	VAR robtarget Openhole_694 := [[468.83, -10.99, 179.55], [0.039839, 0.705984, 0.70118, -0.091361], [0,0,0,0], [9E9, 9E9, 9E9, 9E9, 9E9, 9E9]];
	VAR robtarget Openhole_695 := [[469.79, -10.75, 179.43], [0.042242, 0.705844, 0.700663, -0.095246], [0,0,0,0], [9E9, 9E9, 9E9, 9E9, 9E9, 9E9]];
	VAR robtarget Openhole_696 := [[473.7, -10.06, 178.96], [0.052829, 0.705131, 0.698512, -0.109911], [0,0,0,0], [9E9, 9E9, 9E9, 9E9, 9E9, 9E9]];
	VAR robtarget Openhole_697 := [[478.16, -9.69, 178.47], [0.066049, 0.704015, 0.695989, -0.124897], [0,0,0,0], [9E9, 9E9, 9E9, 9E9, 9E9, 9E9]];
	VAR robtarget Openhole_698 := [[482.14, -9.61, 178.09], [0.078462, 0.70274, 0.693688, -0.137102], [0,0,0,0], [9E9, 9E9, 9E9, 9E9, 9E9, 9E9]];
	VAR robtarget Openhole_699 := [[482.63, -9.62, 178.05], [0.080033, 0.702563, 0.693396, -0.13857], [0,0,0,0], [9E9, 9E9, 9E9, 9E9, 9E9, 9E9]];
	VAR robtarget Openhole_700 := [[494.09, -10.02, 177.18], [0.116014, 0.697525, 0.686428, -0.169755], [0,0,0,0], [9E9, 9E9, 9E9, 9E9, 9E9, 9E9]];
	VAR robtarget Openhole_701 := [[499.58, -10.13, 176.76], [0.132008, 0.694675, 0.682777, -0.183891], [0,0,0,0], [9E9, 9E9, 9E9, 9E9, 9E9, 9E9]];
	VAR robtarget Openhole_702 := [[500.07, -10.12, 176.71], [0.133393, 0.694411, 0.682429, -0.185176], [0,0,0,0], [9E9, 9E9, 9E9, 9E9, 9E9, 9E9]];
	VAR robtarget Openhole_703 := [[503.55, -10.02, 176.36], [0.142648, 0.692569, 0.6799, -0.194257], [0,0,0,0], [9E9, 9E9, 9E9, 9E9, 9E9, 9E9]];
	VAR robtarget Openhole_704 := [[504.33, -10, 176.29], [0.144708, 0.692141, 0.679339, -0.196212], [0,0,0,0], [9E9, 9E9, 9E9, 9E9, 9E9, 9E9]];
	VAR robtarget Openhole_705 := [[509.33, -10, 175.85], [0.183051, 0.683002, 0.683002, -0.183051], [0,0,0,0], [9E9, 9E9, 9E9, 9E9, 9E9, 9E9]];
	VAR robtarget Openhole_706 := [[536.33, -10, 175.77], [0.183051, 0.683002, 0.683002, -0.183051], [0,0,0,0], [9E9, 9E9, 9E9, 9E9, 9E9, 9E9]];
	VAR robtarget Openhole_707 := [[536.33, -10.89, 176.28], [0.183051, 0.683002, 0.683002, -0.183051], [0,0,0,0], [9E9, 9E9, 9E9, 9E9, 9E9, 9E9]];
	VAR robtarget Openhole_708 := [[524.33, -10.89, 176.31], [0.183051, 0.683002, 0.683002, -0.183051], [0,0,0,0], [9E9, 9E9, 9E9, 9E9, 9E9, 9E9]];
	VAR robtarget Openhole_709 := [[509.33, -10.89, 176.36], [0.183051, 0.683002, 0.683002, -0.183051], [0,0,0,0], [9E9, 9E9, 9E9, 9E9, 9E9, 9E9]];
	VAR robtarget Openhole_710 := [[504.39, -10.89, 176.75], [0.147452, 0.691562, 0.680025, -0.19382], [0,0,0,0], [9E9, 9E9, 9E9, 9E9, 9E9, 9E9]];
	VAR robtarget Openhole_711 := [[498.87, -11.14, 177.3], [0.13304, 0.694478, 0.684057, -0.179068], [0,0,0,0], [9E9, 9E9, 9E9, 9E9, 9E9, 9E9]];
	VAR robtarget Openhole_712 := [[497.37, -11.14, 177.42], [0.12885, 0.695268, 0.685077, -0.175125], [0,0,0,0], [9E9, 9E9, 9E9, 9E9, 9E9, 9E9]];
	VAR robtarget Openhole_713 := [[496.87, -11.14, 177.45], [0.127427, 0.69553, 0.685411, -0.173814], [0,0,0,0], [9E9, 9E9, 9E9, 9E9, 9E9, 9E9]];
	VAR robtarget Openhole_714 := [[482.41, -10.79, 178.44], [0.083092, 0.702208, 0.69426, -0.134176], [0,0,0,0], [9E9, 9E9, 9E9, 9E9, 9E9, 9E9]];
	VAR robtarget Openhole_715 := [[481.91, -10.8, 178.48], [0.081533, 0.70239, 0.694546, -0.132689], [0,0,0,0], [9E9, 9E9, 9E9, 9E9, 9E9, 9E9]];
	VAR robtarget Openhole_716 := [[476.44, -10.97, 178.96], [0.064669, 0.704143, 0.69761, -0.115499], [0,0,0,0], [9E9, 9E9, 9E9, 9E9, 9E9, 9E9]];
	VAR robtarget Openhole_717 := [[472.49, -11.44, 179.37], [0.053367, 0.70509, 0.699769, -0.101607], [0,0,0,0], [9E9, 9E9, 9E9, 9E9, 9E9, 9E9]];
	VAR robtarget Openhole_718 := [[471.02, -11.7, 179.53], [0.049411, 0.705378, 0.700549, -0.096078], [0,0,0,0], [9E9, 9E9, 9E9, 9E9, 9E9, 9E9]];
	VAR robtarget Openhole_719 := [[470.53, -11.8, 179.59], [0.048148, 0.705466, 0.700806, -0.094186], [0,0,0,0], [9E9, 9E9, 9E9, 9E9, 9E9, 9E9]];
	VAR robtarget Openhole_720 := [[469.57, -12.03, 179.7], [0.045713, 0.705628, 0.701314, -0.090326], [0,0,0,0], [9E9, 9E9, 9E9, 9E9, 9E9, 9E9]];
	VAR robtarget Openhole_721 := [[468.61, -12.29, 179.81], [0.043403, 0.705773, 0.701812, -0.086369], [0,0,0,0], [9E9, 9E9, 9E9, 9E9, 9E9, 9E9]];
	VAR robtarget Openhole_722 := [[467.66, -12.58, 179.92], [0.041218, 0.705904, 0.702299, -0.08232], [0,0,0,0], [9E9, 9E9, 9E9, 9E9, 9E9, 9E9]];
	VAR robtarget Openhole_723 := [[466.25, -13.07, 180.09], [0.038201, 0.706074, 0.703002, -0.076079], [0,0,0,0], [9E9, 9E9, 9E9, 9E9, 9E9, 9E9]];
	VAR robtarget Openhole_724 := [[465.79, -13.26, 180.15], [0.037278, 0.706123, 0.703229, -0.073951], [0,0,0,0], [9E9, 9E9, 9E9, 9E9, 9E9, 9E9]];
	VAR robtarget Openhole_725 := [[465.33, -13.45, 180.2], [0.036401, 0.706169, 0.703452, -0.071798], [0,0,0,0], [9E9, 9E9, 9E9, 9E9, 9E9, 9E9]];
	VAR robtarget Openhole_726 := [[464.88, -13.66, 180.26], [0.03558, 0.706211, 0.703671, -0.06962], [0,0,0,0], [9E9, 9E9, 9E9, 9E9, 9E9, 9E9]];
	VAR robtarget Openhole_727 := [[463.11, -14.56, 180.47], [0.032691, 0.706351, 0.704495, -0.060722], [0,0,0,0], [9E9, 9E9, 9E9, 9E9, 9E9, 9E9]];
	VAR robtarget Openhole_728 := [[461.82, -15.31, 180.62], [0.030887, 0.706432, 0.70505, -0.053896], [0,0,0,0], [9E9, 9E9, 9E9, 9E9, 9E9, 9E9]];
	VAR robtarget Openhole_729 := [[460.15, -16.4, 180.79], [0.028933, 0.706515, 0.705697, -0.044632], [0,0,0,0], [9E9, 9E9, 9E9, 9E9, 9E9, 9E9]];
	VAR robtarget Openhole_730 := [[459.72, -16.65, 180.82], [0.028341, 0.706539, 0.705839, -0.04233], [0,0,0,0], [9E9, 9E9, 9E9, 9E9, 9E9, 9E9]];
	VAR robtarget Openhole_731 := [[459.27, -16.88, 180.86], [0.027587, 0.706568, 0.70597, -0.040074], [0,0,0,0], [9E9, 9E9, 9E9, 9E9, 9E9, 9E9]];
	VAR robtarget Openhole_732 := [[458.82, -17.08, 180.88], [0.026741, 0.706601, 0.706093, -0.037847], [0,0,0,0], [9E9, 9E9, 9E9, 9E9, 9E9, 9E9]];
	VAR robtarget Openhole_733 := [[458.35, -17.26, 180.91], [0.025788, 0.706636, 0.706207, -0.03566], [0,0,0,0], [9E9, 9E9, 9E9, 9E9, 9E9, 9E9]];
	VAR robtarget Openhole_734 := [[457.88, -17.43, 180.93], [0.024778, 0.706673, 0.706313, -0.033497], [0,0,0,0], [9E9, 9E9, 9E9, 9E9, 9E9, 9E9]];
	VAR robtarget Openhole_735 := [[457.27, -17.6, 180.95], [0.023274, 0.706724, 0.706433, -0.030857], [0,0,0,0], [9E9, 9E9, 9E9, 9E9, 9E9, 9E9]];
	VAR robtarget Openhole_736 := [[454.82, -17.6, 180.99], [0.014998, 0.706948, 0.706747, -0.022558], [0,0,0,0], [9E9, 9E9, 9E9, 9E9, 9E9, 9E9]];
	VAR robtarget Openhole_737 := [[454.9, -18.58, 181.04], [0.018567, 0.706863, 0.706838, -0.019489], [0,0,0,0], [9E9, 9E9, 9E9, 9E9, 9E9, 9E9]];
	VAR robtarget Openhole_738 := [[457.34, -18.58, 181.03], [0.026836, 0.706597, 0.70656, -0.027794], [0,0,0,0], [9E9, 9E9, 9E9, 9E9, 9E9, 9E9]];
	VAR robtarget Openhole_739 := [[457.46, -18.57, 181.03], [0.027232, 0.706582, 0.706544, -0.0282], [0,0,0,0], [9E9, 9E9, 9E9, 9E9, 9E9, 9E9]];
	VAR robtarget Openhole_740 := [[457.96, -18.57, 181.02], [0.028901, 0.706516, 0.706474, -0.029909], [0,0,0,0], [9E9, 9E9, 9E9, 9E9, 9E9, 9E9]];
	VAR robtarget Openhole_741 := [[458.45, -18.46, 181.01], [0.030176, 0.706463, 0.706386, -0.031929], [0,0,0,0], [9E9, 9E9, 9E9, 9E9, 9E9, 9E9]];
	VAR robtarget Openhole_742 := [[459.42, -18.22, 180.98], [0.032613, 0.706354, 0.706188, -0.036029], [0,0,0,0], [9E9, 9E9, 9E9, 9E9, 9E9, 9E9]];
	VAR robtarget Openhole_743 := [[460.37, -17.92, 180.94], [0.03481, 0.706249, 0.70596, -0.040251], [0,0,0,0], [9E9, 9E9, 9E9, 9E9, 9E9, 9E9]];
	VAR robtarget Openhole_744 := [[460.84, -17.74, 180.92], [0.035759, 0.706202, 0.705833, -0.042429], [0,0,0,0], [9E9, 9E9, 9E9, 9E9, 9E9, 9E9]];
	VAR robtarget Openhole_745 := [[461.3, -17.54, 180.89], [0.036653, 0.706156, 0.705697, -0.044628], [0,0,0,0], [9E9, 9E9, 9E9, 9E9, 9E9, 9E9]];
	VAR robtarget Openhole_746 := [[462.19, -17.09, 180.82], [0.038087, 0.70608, 0.705397, -0.049141], [0,0,0,0], [9E9, 9E9, 9E9, 9E9, 9E9, 9E9]];
	VAR robtarget Openhole_747 := [[463.94, -16.14, 180.66], [0.040777, 0.70593, 0.70471, -0.058174], [0,0,0,0], [9E9, 9E9, 9E9, 9E9, 9E9, 9E9]];
	VAR robtarget Openhole_748 := [[464.83, -15.7, 180.57], [0.042243, 0.705844, 0.704328, -0.062628], [0,0,0,0], [9E9, 9E9, 9E9, 9E9, 9E9, 9E9]];
	VAR robtarget Openhole_749 := [[465.73, -15.28, 180.47], [0.043835, 0.705747, 0.703924, -0.067018], [0,0,0,0], [9E9, 9E9, 9E9, 9E9, 9E9, 9E9]];
	VAR robtarget Openhole_750 := [[466.19, -15.08, 180.42], [0.044689, 0.705693, 0.703714, -0.069185], [0,0,0,0], [9E9, 9E9, 9E9, 9E9, 9E9, 9E9]];
	VAR robtarget Openhole_751 := [[466.65, -14.89, 180.37], [0.045584, 0.705636, 0.7035, -0.07133], [0,0,0,0], [9E9, 9E9, 9E9, 9E9, 9E9, 9E9]];
	VAR robtarget Openhole_752 := [[467.12, -14.71, 180.32], [0.046532, 0.705574, 0.703282, -0.073447], [0,0,0,0], [9E9, 9E9, 9E9, 9E9, 9E9, 9E9]];
	VAR robtarget Openhole_753 := [[467.58, -14.54, 180.27], [0.047528, 0.705508, 0.703061, -0.075537], [0,0,0,0], [9E9, 9E9, 9E9, 9E9, 9E9, 9E9]];
	VAR robtarget Openhole_754 := [[468.53, -14.24, 180.18], [0.049641, 0.705362, 0.702607, -0.079642], [0,0,0,0], [9E9, 9E9, 9E9, 9E9, 9E9, 9E9]];
	VAR robtarget Openhole_755 := [[469.49, -13.97, 180.08], [0.0519, 0.7052, 0.702142, -0.083648], [0,0,0,0], [9E9, 9E9, 9E9, 9E9, 9E9, 9E9]];
	VAR robtarget Openhole_756 := [[470.46, -13.73, 179.98], [0.054271, 0.705021, 0.701664, -0.087567], [0,0,0,0], [9E9, 9E9, 9E9, 9E9, 9E9, 9E9]];
	VAR robtarget Openhole_757 := [[470.94, -13.62, 179.94], [0.055498, 0.704925, 0.701421, -0.089491], [0,0,0,0], [9E9, 9E9, 9E9, 9E9, 9E9, 9E9]];
	VAR robtarget Openhole_758 := [[471.92, -13.42, 179.84], [0.058039, 0.704721, 0.700929, -0.093267], [0,0,0,0], [9E9, 9E9, 9E9, 9E9, 9E9, 9E9]];
	VAR robtarget Openhole_759 := [[475.87, -12.91, 179.5], [0.069183, 0.703714, 0.698901, -0.107409], [0,0,0,0], [9E9, 9E9, 9E9, 9E9, 9E9, 9E9]];
	VAR robtarget Openhole_760 := [[480.85, -12.71, 179.15], [0.084353, 0.702057, 0.69626, -0.12338], [0,0,0,0], [9E9, 9E9, 9E9, 9E9, 9E9, 9E9]];
	VAR robtarget Openhole_761 := [[482.35, -12.7, 179.05], [0.088996, 0.701484, 0.69544, -0.127919], [0,0,0,0], [9E9, 9E9, 9E9, 9E9, 9E9, 9E9]];
	VAR robtarget Openhole_762 := [[482.85, -12.7, 179.02], [0.090547, 0.701285, 0.695164, -0.12941], [0,0,0,0], [9E9, 9E9, 9E9, 9E9, 9E9, 9E9]];
	VAR robtarget Openhole_763 := [[495.33, -12.89, 178.35], [0.12834, 0.695362, 0.687731, -0.164398], [0,0,0,0], [9E9, 9E9, 9E9, 9E9, 9E9, 9E9]];
	VAR robtarget Openhole_764 := [[495.83, -12.89, 178.32], [0.129759, 0.695099, 0.687406, -0.165751], [0,0,0,0], [9E9, 9E9, 9E9, 9E9, 9E9, 9E9]];
	VAR robtarget Openhole_765 := [[501.81, -12.75, 177.89], [0.145951, 0.69188, 0.683309, -0.181905], [0,0,0,0], [9E9, 9E9, 9E9, 9E9, 9E9, 9E9]];
	VAR robtarget Openhole_766 := [[504.33, -12.58, 177.65], [0.152252, 0.690521, 0.681443, -0.188774], [0,0,0,0], [9E9, 9E9, 9E9, 9E9, 9E9, 9E9]];
	VAR robtarget Openhole_767 := [[509.33, -12.58, 177.34], [0.183051, 0.683002, 0.683002, -0.183051], [0,0,0,0], [9E9, 9E9, 9E9, 9E9, 9E9, 9E9]];
	VAR robtarget Openhole_768 := [[536.33, -12.58, 177.26], [0.183051, 0.683002, 0.683002, -0.183051], [0,0,0,0], [9E9, 9E9, 9E9, 9E9, 9E9, 9E9]];
	VAR robtarget Openhole_769 := [[536.34, -16.49, 179.51], [0.183051, 0.683002, 0.683002, -0.183051], [0,0,0,0], [9E9, 9E9, 9E9, 9E9, 9E9, 9E9]];
	VAR robtarget Openhole_770 := [[509.34, -16.49, 179.6], [0.183051, 0.683002, 0.683002, -0.183051], [0,0,0,0], [9E9, 9E9, 9E9, 9E9, 9E9, 9E9]];
	VAR robtarget Openhole_771 := [[504.34, -16.49, 179.72], [0.163682, 0.687901, 0.684485, -0.177427], [0,0,0,0], [9E9, 9E9, 9E9, 9E9, 9E9, 9E9]];
	VAR robtarget Openhole_772 := [[497.74, -16.81, 180.03], [0.146949, 0.691669, 0.688969, -0.159127], [0,0,0,0], [9E9, 9E9, 9E9, 9E9, 9E9, 9E9]];
	VAR robtarget Openhole_773 := [[491.74, -16.89, 180.19], [0.130322, 0.694994, 0.692656, -0.142222], [0,0,0,0], [9E9, 9E9, 9E9, 9E9, 9E9, 9E9]];
	VAR robtarget Openhole_774 := [[491.24, -16.89, 180.2], [0.12888, 0.695263, 0.692947, -0.140799], [0,0,0,0], [9E9, 9E9, 9E9, 9E9, 9E9, 9E9]];
	VAR robtarget Openhole_775 := [[478.25, -16.73, 180.42], [0.08917, 0.701462, 0.699653, -0.102403], [0,0,0,0], [9E9, 9E9, 9E9, 9E9, 9E9, 9E9]];
	VAR robtarget Openhole_776 := [[477.75, -16.74, 180.44], [0.087603, 0.701659, 0.69988, -0.100837], [0,0,0,0], [9E9, 9E9, 9E9, 9E9, 9E9, 9E9]];
	VAR robtarget Openhole_777 := [[472.25, -16.88, 180.59], [0.070529, 0.703581, 0.702227, -0.082932], [0,0,0,0], [9E9, 9E9, 9E9, 9E9, 9E9, 9E9]];
	VAR robtarget Openhole_778 := [[471.26, -16.95, 180.62], [0.067552, 0.703873, 0.702627, -0.079465], [0,0,0,0], [9E9, 9E9, 9E9, 9E9, 9E9, 9E9]];
	VAR robtarget Openhole_779 := [[470.26, -17.06, 180.67], [0.064687, 0.704142, 0.703023, -0.075881], [0,0,0,0], [9E9, 9E9, 9E9, 9E9, 9E9, 9E9]];
	VAR robtarget Openhole_780 := [[468.29, -17.35, 180.76], [0.05919, 0.704625, 0.703785, -0.06846], [0,0,0,0], [9E9, 9E9, 9E9, 9E9, 9E9, 9E9]];
	VAR robtarget Openhole_781 := [[467.79, -17.44, 180.78], [0.057875, 0.704734, 0.703968, -0.06655], [0,0,0,0], [9E9, 9E9, 9E9, 9E9, 9E9, 9E9]];
	VAR robtarget Openhole_782 := [[467.31, -17.54, 180.8], [0.056598, 0.704838, 0.704149, -0.064606], [0,0,0,0], [9E9, 9E9, 9E9, 9E9, 9E9, 9E9]];
	VAR robtarget Openhole_783 := [[465.37, -18.02, 180.91], [0.05178, 0.705208, 0.704838, -0.056602], [0,0,0,0], [9E9, 9E9, 9E9, 9E9, 9E9, 9E9]];
	VAR robtarget Openhole_784 := [[464.4, -18.28, 180.95], [0.049485, 0.705373, 0.705155, -0.052504], [0,0,0,0], [9E9, 9E9, 9E9, 9E9, 9E9, 9E9]];
	VAR robtarget Openhole_785 := [[463.43, -18.53, 180.99], [0.047088, 0.705537, 0.705445, -0.048449], [0,0,0,0], [9E9, 9E9, 9E9, 9E9, 9E9, 9E9]];
	VAR robtarget Openhole_786 := [[460.01, -19.25, 181.08], [0.038081, 0.706081, 0.706264, -0.034517], [0,0,0,0], [9E9, 9E9, 9E9, 9E9, 9E9, 9E9]];
	VAR robtarget Openhole_787 := [[458.03, -19.56, 181.11], [0.03249, 0.70636, 0.706599, -0.026789], [0,0,0,0], [9E9, 9E9, 9E9, 9E9, 9E9, 9E9]];
	VAR robtarget Openhole_788 := [[457.29, -19.61, 181.11], [0.030166, 0.706463, 0.706696, -0.024105], [0,0,0,0], [9E9, 9E9, 9E9, 9E9, 9E9, 9E9]];
	VAR robtarget Openhole_789 := [[454.85, -19.61, 181.09], [0.021903, 0.706767, 0.70693, -0.015793], [0,0,0,0], [9E9, 9E9, 9E9, 9E9, 9E9, 9E9]];
	VAR robtarget Openhole_790 := [[454.65, -20.66, 181.14], [0.024813, 0.706671, 0.707012, -0.011567], [0,0,0,0], [9E9, 9E9, 9E9, 9E9, 9E9, 9E9]];
	VAR robtarget Openhole_791 := [[457.1, -20.66, 181.18], [0.033072, 0.706333, 0.706827, -0.019887], [0,0,0,0], [9E9, 9E9, 9E9, 9E9, 9E9, 9E9]];
	VAR robtarget Openhole_792 := [[457.64, -20.63, 181.19], [0.034803, 0.70625, 0.70677, -0.02182], [0,0,0,0], [9E9, 9E9, 9E9, 9E9, 9E9, 9E9]];
	VAR robtarget Openhole_793 := [[458.63, -20.47, 181.19], [0.037562, 0.706108, 0.706639, -0.025721], [0,0,0,0], [9E9, 9E9, 9E9, 9E9, 9E9, 9E9]];
	VAR robtarget Openhole_794 := [[459.13, -20.43, 181.19], [0.039097, 0.706025, 0.70657, -0.027546], [0,0,0,0], [9E9, 9E9, 9E9, 9E9, 9E9, 9E9]];
	VAR robtarget Openhole_795 := [[460.13, -20.37, 181.2], [0.042255, 0.705843, 0.706422, -0.031109], [0,0,0,0], [9E9, 9E9, 9E9, 9E9, 9E9, 9E9]];
	VAR robtarget Openhole_796 := [[461.63, -20.35, 181.22], [0.047187, 0.705531, 0.706177, -0.036242], [0,0,0,0], [9E9, 9E9, 9E9, 9E9, 9E9, 9E9]];
	VAR robtarget Openhole_797 := [[462.63, -20.37, 181.23], [0.05057, 0.705296, 0.706, -0.039549], [0,0,0,0], [9E9, 9E9, 9E9, 9E9, 9E9, 9E9]];
	VAR robtarget Openhole_798 := [[464.13, -20.42, 181.26], [0.055739, 0.704906, 0.705713, -0.04437], [0,0,0,0], [9E9, 9E9, 9E9, 9E9, 9E9, 9E9]];
	VAR robtarget Openhole_799 := [[480.61, -20.9, 181.63], [0.109951, 0.698506, 0.700524, -0.096261], [0,0,0,0], [9E9, 9E9, 9E9, 9E9, 9E9, 9E9]];
	VAR robtarget Openhole_800 := [[489.11, -20.98, 181.81], [0.135434, 0.694016, 0.696533, -0.121825], [0,0,0,0], [9E9, 9E9, 9E9, 9E9, 9E9, 9E9]];
	VAR robtarget Openhole_801 := [[489.61, -20.98, 181.82], [0.136869, 0.693734, 0.696273, -0.123302], [0,0,0,0], [9E9, 9E9, 9E9, 9E9, 9E9, 9E9]];
	VAR robtarget Openhole_802 := [[499.61, -20.8, 181.92], [0.163935, 0.687841, 0.690534, -0.152193], [0,0,0,0], [9E9, 9E9, 9E9, 9E9, 9E9, 9E9]];
	VAR robtarget Openhole_803 := [[504.35, -20.6, 181.89], [0.175641, 0.684946, 0.687477, -0.165454], [0,0,0,0], [9E9, 9E9, 9E9, 9E9, 9E9, 9E9]];
	VAR robtarget Openhole_804 := [[509.35, -20.6, 181.97], [0.183051, 0.683002, 0.683002, -0.183051], [0,0,0,0], [9E9, 9E9, 9E9, 9E9, 9E9, 9E9]];
	VAR robtarget Openhole_805 := [[536.35, -20.6, 181.88], [0.183051, 0.683002, 0.683002, -0.183051], [0,0,0,0], [9E9, 9E9, 9E9, 9E9, 9E9, 9E9]];
	VAR robtarget Openhole_806 := [[536.35, -22.17, 182.79], [0.183051, 0.683002, 0.683002, -0.183051], [0,0,0,0], [9E9, 9E9, 9E9, 9E9, 9E9, 9E9]];
	VAR robtarget Openhole_807 := [[509.35, -22.17, 182.88], [0.183051, 0.683002, 0.683002, -0.183051], [0,0,0,0], [9E9, 9E9, 9E9, 9E9, 9E9, 9E9]];
	VAR robtarget Openhole_808 := [[504.35, -22.17, 182.72], [0.180212, 0.683757, 0.688569, -0.160849], [0,0,0,0], [9E9, 9E9, 9E9, 9E9, 9E9, 9E9]];
	VAR robtarget Openhole_809 := [[494.58, -22.52, 182.58], [0.155534, 0.689789, 0.694498, -0.132936], [0,0,0,0], [9E9, 9E9, 9E9, 9E9, 9E9, 9E9]];
	VAR robtarget Openhole_810 := [[485.58, -22.61, 182.31], [0.130261, 0.695005, 0.699101, -0.1061], [0,0,0,0], [9E9, 9E9, 9E9, 9E9, 9E9, 9E9]];
	VAR robtarget Openhole_811 := [[485.08, -22.61, 182.29], [0.128791, 0.695279, 0.699331, -0.104576], [0,0,0,0], [9E9, 9E9, 9E9, 9E9, 9E9, 9E9]];
	VAR robtarget Openhole_812 := [[471.59, -22.42, 181.79], [0.086679, 0.701774, 0.704346, -0.062427], [0,0,0,0], [9E9, 9E9, 9E9, 9E9, 9E9, 9E9]];
	VAR robtarget Openhole_813 := [[465.61, -22.1, 181.54], [0.066221, 0.703999, 0.705755, -0.043698], [0,0,0,0], [9E9, 9E9, 9E9, 9E9, 9E9, 9E9]];
	VAR robtarget Openhole_814 := [[461.64, -21.66, 181.37], [0.051628, 0.70522, 0.70639, -0.031841], [0,0,0,0], [9E9, 9E9, 9E9, 9E9, 9E9, 9E9]];
	VAR robtarget Openhole_815 := [[460.14, -21.53, 181.32], [0.046218, 0.705595, 0.706582, -0.02723], [0,0,0,0], [9E9, 9E9, 9E9, 9E9, 9E9, 9E9]];
	VAR robtarget Openhole_816 := [[459.64, -21.51, 181.31], [0.044462, 0.705708, 0.706642, -0.02563], [0,0,0,0], [9E9, 9E9, 9E9, 9E9, 9E9, 9E9]];
	VAR robtarget Openhole_817 := [[459.14, -21.49, 181.29], [0.042747, 0.705813, 0.7067, -0.02398], [0,0,0,0], [9E9, 9E9, 9E9, 9E9, 9E9, 9E9]];
	VAR robtarget Openhole_818 := [[458.64, -21.5, 181.28], [0.041075, 0.705913, 0.706756, -0.022282], [0,0,0,0], [9E9, 9E9, 9E9, 9E9, 9E9, 9E9]];
	VAR robtarget Openhole_819 := [[458.14, -21.51, 181.27], [0.039453, 0.706005, 0.706809, -0.020533], [0,0,0,0], [9E9, 9E9, 9E9, 9E9, 9E9, 9E9]];
	VAR robtarget Openhole_820 := [[457.66, -21.63, 181.27], [0.038219, 0.706073, 0.706865, -0.018484], [0,0,0,0], [9E9, 9E9, 9E9, 9E9, 9E9, 9E9]];
	VAR robtarget Openhole_821 := [[456.8, -21.6, 181.25], [0.035247, 0.706228, 0.706933, -0.015657], [0,0,0,0], [9E9, 9E9, 9E9, 9E9, 9E9, 9E9]];
	VAR robtarget Openhole_822 := [[454.35, -21.6, 181.19], [0.02699, 0.706592, 0.707069, -0.007329], [0,0,0,0], [9E9, 9E9, 9E9, 9E9, 9E9, 9E9]];
	VAR robtarget Openhole_823 := [[453.91, -22.56, 181.22], [0.028711, 0.706524, 0.707102, -0.002571], [0,0,0,0], [9E9, 9E9, 9E9, 9E9, 9E9, 9E9]];
	VAR robtarget Openhole_824 := [[456.36, -22.56, 181.3], [0.036968, 0.70614, 0.707023, -0.010907], [0,0,0,0], [9E9, 9E9, 9E9, 9E9, 9E9, 9E9]];
	VAR robtarget Openhole_825 := [[456.89, -22.57, 181.32], [0.038832, 0.70604, 0.706993, -0.012682], [0,0,0,0], [9E9, 9E9, 9E9, 9E9, 9E9, 9E9]];
	VAR robtarget Openhole_826 := [[457.39, -22.58, 181.34], [0.040526, 0.705945, 0.706961, -0.014366], [0,0,0,0], [9E9, 9E9, 9E9, 9E9, 9E9, 9E9]];
	VAR robtarget Openhole_827 := [[458.89, -22.62, 181.39], [0.045703, 0.705628, 0.706843, -0.0193], [0,0,0,0], [9E9, 9E9, 9E9, 9E9, 9E9, 9E9]];
	VAR robtarget Openhole_828 := [[459.89, -22.67, 181.43], [0.049215, 0.705392, 0.706749, -0.022505], [0,0,0,0], [9E9, 9E9, 9E9, 9E9, 9E9, 9E9]];
	VAR robtarget Openhole_829 := [[465.84, -23.34, 181.75], [0.071117, 0.703521, 0.705956, -0.040325], [0,0,0,0], [9E9, 9E9, 9E9, 9E9, 9E9, 9E9]];
	VAR robtarget Openhole_830 := [[472.83, -23.6, 182.1], [0.094484, 0.700766, 0.704335, -0.062552], [0,0,0,0], [9E9, 9E9, 9E9, 9E9, 9E9, 9E9]];
	VAR robtarget Openhole_831 := [[480.32, -23.66, 182.44], [0.117891, 0.69721, 0.701805, -0.086425], [0,0,0,0], [9E9, 9E9, 9E9, 9E9, 9E9, 9E9]];
	VAR robtarget Openhole_832 := [[480.82, -23.66, 182.46], [0.119401, 0.696953, 0.70161, -0.087997], [0,0,0,0], [9E9, 9E9, 9E9, 9E9, 9E9, 9E9]];
	VAR robtarget Openhole_833 := [[481.32, -23.66, 182.49], [0.120908, 0.696693, 0.701411, -0.089565], [0,0,0,0], [9E9, 9E9, 9E9, 9E9, 9E9, 9E9]];
	VAR robtarget Openhole_834 := [[481.82, -23.66, 182.51], [0.122405, 0.696432, 0.70121, -0.091132], [0,0,0,0], [9E9, 9E9, 9E9, 9E9, 9E9, 9E9]];
	VAR robtarget Openhole_835 := [[495.81, -23.48, 183.05], [0.161772, 0.688353, 0.694388, -0.133511], [0,0,0,0], [9E9, 9E9, 9E9, 9E9, 9E9, 9E9]];
	VAR robtarget Openhole_836 := [[504.35, -23.14, 183.24], [0.183021, 0.683011, 0.689226, -0.158013], [0,0,0,0], [9E9, 9E9, 9E9, 9E9, 9E9, 9E9]];
	VAR robtarget Openhole_837 := [[509.35, -23.14, 183.44], [0.183051, 0.683002, 0.683002, -0.183051], [0,0,0,0], [9E9, 9E9, 9E9, 9E9, 9E9, 9E9]];
	VAR robtarget Openhole_838 := [[536.35, -23.14, 183.35], [0.183051, 0.683002, 0.683002, -0.183051], [0,0,0,0], [9E9, 9E9, 9E9, 9E9, 9E9, 9E9]];
	VAR robtarget Openhole_839 := [[536.35, -24.03, 183.87], [0.183051, 0.683002, 0.683002, -0.183051], [0,0,0,0], [9E9, 9E9, 9E9, 9E9, 9E9, 9E9]];
	VAR robtarget Openhole_840 := [[509.35, -24.03, 183.95], [0.183051, 0.683002, 0.683002, -0.183051], [0,0,0,0], [9E9, 9E9, 9E9, 9E9, 9E9, 9E9]];
	VAR robtarget Openhole_841 := [[504.35, -24.03, 183.71], [0.18561, 0.682311, 0.689821, -0.155392], [0,0,0,0], [9E9, 9E9, 9E9, 9E9, 9E9, 9E9]];
	VAR robtarget Openhole_842 := [[493.5, -24.43, 183.36], [0.158367, 0.689144, 0.696158, -0.123954], [0,0,0,0], [9E9, 9E9, 9E9, 9E9, 9E9, 9E9]];
	VAR robtarget Openhole_843 := [[477.02, -24.66, 182.56], [0.111028, 0.698336, 0.703365, -0.072646], [0,0,0,0], [9E9, 9E9, 9E9, 9E9, 9E9, 9E9]];
	VAR robtarget Openhole_844 := [[473.02, -24.68, 182.35], [0.098621, 0.700196, 0.704587, -0.059638], [0,0,0,0], [9E9, 9E9, 9E9, 9E9, 9E9, 9E9]];
	VAR robtarget Openhole_845 := [[472.53, -24.68, 182.32], [0.097043, 0.700416, 0.704724, -0.058005], [0,0,0,0], [9E9, 9E9, 9E9, 9E9, 9E9, 9E9]];
	VAR robtarget Openhole_846 := [[465.04, -24.53, 181.89], [0.072456, 0.703385, 0.706306, -0.033633], [0,0,0,0], [9E9, 9E9, 9E9, 9E9, 9E9, 9E9]];
	VAR robtarget Openhole_847 := [[458.58, -23.97, 181.5], [0.04919, 0.705394, 0.706975, -0.013663], [0,0,0,0], [9E9, 9E9, 9E9, 9E9, 9E9, 9E9]];
	VAR robtarget Openhole_848 := [[457.08, -23.91, 181.42], [0.04397, 0.705738, 0.707052, -0.008779], [0,0,0,0], [9E9, 9E9, 9E9, 9E9, 9E9, 9E9]];
	VAR robtarget Openhole_849 := [[456.08, -23.86, 181.37], [0.040449, 0.705949, 0.707085, -0.005552], [0,0,0,0], [9E9, 9E9, 9E9, 9E9, 9E9, 9E9]];
	VAR robtarget Openhole_850 := [[455.52, -23.79, 181.34], [0.038313, 0.706068, 0.707096, -0.003893], [0,0,0,0], [9E9, 9E9, 9E9, 9E9, 9E9, 9E9]];
	VAR robtarget Openhole_851 := [[453.07, -23.79, 181.23], [0.030052, 0.706468, 0.707093, 0.004452], [0,0,0,0], [9E9, 9E9, 9E9, 9E9, 9E9, 9E9]];
	VAR robtarget Openhole_852 := [[451.65, -25.14, 181.2], [0.029798, 0.706479, 0.70697, 0.013908], [0,0,0,0], [9E9, 9E9, 9E9, 9E9, 9E9, 9E9]];
	VAR robtarget Openhole_853 := [[454.1, -25.14, 181.34], [0.038071, 0.706081, 0.707085, 0.005557], [0,0,0,0], [9E9, 9E9, 9E9, 9E9, 9E9, 9E9]];
	VAR robtarget Openhole_854 := [[454.68, -25.32, 181.38], [0.040677, 0.705936, 0.707094, 0.004175], [0,0,0,0], [9E9, 9E9, 9E9, 9E9, 9E9, 9E9]];
	VAR robtarget Openhole_855 := [[455.18, -25.38, 181.42], [0.042528, 0.705827, 0.707102, 0.002663], [0,0,0,0], [9E9, 9E9, 9E9, 9E9, 9E9, 9E9]];
	VAR robtarget Openhole_856 := [[455.68, -25.42, 181.45], [0.044346, 0.705715, 0.707106, 0.001116], [0,0,0,0], [9E9, 9E9, 9E9, 9E9, 9E9, 9E9]];
	VAR robtarget Openhole_857 := [[465.15, -25.83, 182.1], [0.077135, 0.702887, 0.706486, -0.029619], [0,0,0,0], [9E9, 9E9, 9E9, 9E9, 9E9, 9E9]];
	VAR robtarget Openhole_858 := [[467.64, -25.85, 182.26], [0.085306, 0.701942, 0.70609, -0.037909], [0,0,0,0], [9E9, 9E9, 9E9, 9E9, 9E9, 9E9]];
	VAR robtarget Openhole_859 := [[468.14, -25.85, 182.3], [0.086911, 0.701745, 0.705998, -0.03958], [0,0,0,0], [9E9, 9E9, 9E9, 9E9, 9E9, 9E9]];
	VAR robtarget Openhole_860 := [[491.1, -25.41, 183.63], [0.154736, 0.689969, 0.697881, -0.113853], [0,0,0,0], [9E9, 9E9, 9E9, 9E9, 9E9, 9E9]];
	VAR robtarget Openhole_861 := [[502.58, -25, 184.12], [0.18397, 0.682755, 0.691498, -0.147751], [0,0,0,0], [9E9, 9E9, 9E9, 9E9, 9E9, 9E9]];
	VAR robtarget Openhole_862 := [[504.36, -24.92, 184.18], [0.188175, 0.681609, 0.690402, -0.152792], [0,0,0,0], [9E9, 9E9, 9E9, 9E9, 9E9, 9E9]];
	VAR robtarget Openhole_863 := [[509.36, -24.92, 184.46], [0.183051, 0.683002, 0.683002, -0.183051], [0,0,0,0], [9E9, 9E9, 9E9, 9E9, 9E9, 9E9]];
	VAR robtarget Openhole_864 := [[536.36, -24.92, 184.38], [0.183051, 0.683002, 0.683002, -0.183051], [0,0,0,0], [9E9, 9E9, 9E9, 9E9, 9E9, 9E9]];
	VAR robtarget Openhole_865 := [[536.36, -25.98, 184.99], [0.183051, 0.683002, 0.683002, -0.183051], [0,0,0,0], [9E9, 9E9, 9E9, 9E9, 9E9, 9E9]];
	VAR robtarget Openhole_866 := [[509.36, -25.98, 185.07], [0.183051, 0.683002, 0.683002, -0.183051], [0,0,0,0], [9E9, 9E9, 9E9, 9E9, 9E9, 9E9]];
	VAR robtarget Openhole_867 := [[504.36, -25.98, 184.74], [0.191223, 0.68076, 0.69108, -0.149694], [0,0,0,0], [9E9, 9E9, 9E9, 9E9, 9E9, 9E9]];
	VAR robtarget Openhole_868 := [[492.57, -26.46, 184.15], [0.16198, 0.688304, 0.697695, -0.114986], [0,0,0,0], [9E9, 9E9, 9E9, 9E9, 9E9, 9E9]];
	VAR robtarget Openhole_869 := [[471.63, -27.19, 182.81], [0.102436, 0.699648, 0.705562, -0.046716], [0,0,0,0], [9E9, 9E9, 9E9, 9E9, 9E9, 9E9]];
	VAR robtarget Openhole_870 := [[456.18, -27.73, 181.63], [0.053821, 0.705056, 0.70707, 0.007227], [0,0,0,0], [9E9, 9E9, 9E9, 9E9, 9E9, 9E9]];
	VAR robtarget Openhole_871 := [[455.68, -27.74, 181.59], [0.052186, 0.705178, 0.70705, 0.008964], [0,0,0,0], [9E9, 9E9, 9E9, 9E9, 9E9, 9E9]];
	VAR robtarget Openhole_872 := [[454.69, -27.73, 181.51], [0.048791, 0.705421, 0.706999, 0.012318], [0,0,0,0], [9E9, 9E9, 9E9, 9E9, 9E9, 9E9]];
	VAR robtarget Openhole_873 := [[454.19, -27.71, 181.47], [0.047048, 0.70554, 0.706969, 0.013948], [0,0,0,0], [9E9, 9E9, 9E9, 9E9, 9E9, 9E9]];
	VAR robtarget Openhole_874 := [[452.7, -27.62, 181.34], [0.041726, 0.705875, 0.706858, 0.01875], [0,0,0,0], [9E9, 9E9, 9E9, 9E9, 9E9, 9E9]];
	VAR robtarget Openhole_875 := [[448.72, -27.39, 181.01], [0.02747, 0.706573, 0.706403, 0.031532], [0,0,0,0], [9E9, 9E9, 9E9, 9E9, 9E9, 9E9]];
	VAR robtarget Openhole_876 := [[448.22, -27.39, 180.97], [0.025771, 0.706637, 0.706326, 0.033221], [0,0,0,0], [9E9, 9E9, 9E9, 9E9, 9E9, 9E9]];
	VAR robtarget Openhole_877 := [[447.72, -27.4, 180.93], [0.024121, 0.706695, 0.706242, 0.034957], [0,0,0,0], [9E9, 9E9, 9E9, 9E9, 9E9, 9E9]];
	VAR robtarget Openhole_878 := [[447.22, -27.43, 180.89], [0.022509, 0.706748, 0.706152, 0.036728], [0,0,0,0], [9E9, 9E9, 9E9, 9E9, 9E9, 9E9]];
	VAR robtarget Openhole_879 := [[445.74, -27.57, 180.76], [0.017922, 0.70688, 0.705843, 0.04225], [0,0,0,0], [9E9, 9E9, 9E9, 9E9, 9E9, 9E9]];
	VAR robtarget Openhole_880 := [[442.28, -28.03, 180.45], [0.007722, 0.707065, 0.704928, 0.055465], [0,0,0,0], [9E9, 9E9, 9E9, 9E9, 9E9, 9E9]];
	VAR robtarget Openhole_881 := [[441.3, -28.17, 180.35], [0.004843, 0.70709, 0.704621, 0.059244], [0,0,0,0], [9E9, 9E9, 9E9, 9E9, 9E9, 9E9]];
	VAR robtarget Openhole_882 := [[438.84, -28.58, 180.1], [-0.002112, 0.707104, 0.703751, 0.068808], [0,0,0,0], [9E9, 9E9, 9E9, 9E9, 9E9, 9E9]];
	VAR robtarget Openhole_883 := [[437.86, -28.76, 179.99], [-0.004844, 0.70709, 0.703366, 0.072642], [0,0,0,0], [9E9, 9E9, 9E9, 9E9, 9E9, 9E9]];
	VAR robtarget Openhole_884 := [[430.07, -30.27, 178.98], [-0.026109, 0.706625, 0.699566, 0.102992], [0,0,0,0], [9E9, 9E9, 9E9, 9E9, 9E9, 9E9]];
	VAR robtarget Openhole_885 := [[425.17, -30.94, 178.29], [-0.04023, 0.705961, 0.696745, 0.120609], [0,0,0,0], [9E9, 9E9, 9E9, 9E9, 9E9, 9E9]];
	VAR robtarget Openhole_886 := [[420.22, -31.24, 177.64], [-0.055453, 0.704929, 0.693776, 0.136657], [0,0,0,0], [9E9, 9E9, 9E9, 9E9, 9E9, 9E9]];
	VAR robtarget Openhole_887 := [[418.24, -31.27, 177.4], [-0.061797, 0.704401, 0.692572, 0.142633], [0,0,0,0], [9E9, 9E9, 9E9, 9E9, 9E9, 9E9]];
	VAR robtarget Openhole_888 := [[417.74, -31.27, 177.34], [-0.063397, 0.704259, 0.69227, 0.144091], [0,0,0,0], [9E9, 9E9, 9E9, 9E9, 9E9, 9E9]];
	VAR robtarget Openhole_889 := [[411.78, -31.03, 176.72], [-0.082989, 0.70222, 0.688647, 0.160517], [0,0,0,0], [9E9, 9E9, 9E9, 9E9, 9E9, 9E9]];
	VAR robtarget Openhole_890 := [[397.86, -29.96, 175.65], [-0.127585, 0.695501, 0.679899, 0.194262], [0,0,0,0], [9E9, 9E9, 9E9, 9E9, 9E9, 9E9]];
	VAR robtarget Openhole_891 := [[394.33, -29.87, 175.32], [-0.137648, 0.69358, 0.677426, 0.202716], [0,0,0,0], [9E9, 9E9, 9E9, 9E9, 9E9, 9E9]];
	VAR robtarget Openhole_892 := [[389.33, -29.87, 174.8], [-0.151079, 0.690779, 0.673786, 0.214504], [0,0,0,0], [9E9, 9E9, 9E9, 9E9, 9E9, 9E9]];
	VAR robtarget Openhole_893 := [[362.33, -29.87, 174.88], [-0.183051, 0.683002, 0.683002, 0.183051], [0,0,0,0], [9E9, 9E9, 9E9, 9E9, 9E9, 9E9]];
	VAR robtarget Openhole_894 := [[361.4, -38.7, 169.79], [-0.183051, 0.683002, 0.683002, 0.183051], [0,0,0,0], [9E9, 9E9, 9E9, 9E9, 9E9, 9E9]];
	VAR robtarget Openhole_895 := [[389.31, -38.7, 169.7], [-0.126057, 0.69578, 0.66558, 0.238752], [0,0,0,0], [9E9, 9E9, 9E9, 9E9, 9E9, 9E9]];
	VAR robtarget Openhole_896 := [[480.22, -38.7, 186.9], [0.164843, 0.687624, 0.706095, -0.037823], [0,0,0,0], [9E9, 9E9, 9E9, 9E9, 9E9, 9E9]];
	VAR robtarget Openhole_897 := [[488.07, -37.66, 188], [0.183568, 0.682864, 0.703974, -0.066484], [0,0,0,0], [9E9, 9E9, 9E9, 9E9, 9E9, 9E9]];
	VAR robtarget Openhole_898 := [[498.44, -36.73, 189.42], [0.207576, 0.675953, 0.699846, -0.101074], [0,0,0,0], [9E9, 9E9, 9E9, 9E9, 9E9, 9E9]];
	VAR robtarget Openhole_899 := [[504.37, -36.35, 190.23], [0.220669, 0.671792, 0.696955, -0.119388], [0,0,0,0], [9E9, 9E9, 9E9, 9E9, 9E9, 9E9]];
	VAR robtarget Openhole_900 := [[504.37, -36.35, 190.23], [0.220681, 0.671789, 0.696952, -0.119405], [0,0,0,0], [9E9, 9E9, 9E9, 9E9, 9E9, 9E9]];
	VAR robtarget Openhole_901 := [[509.38, -36.35, 191.06], [0.183051, 0.683002, 0.683002, -0.183051], [0,0,0,0], [9E9, 9E9, 9E9, 9E9, 9E9, 9E9]];
	VAR robtarget Openhole_902 := [[536.38, -36.35, 190.98], [0.183051, 0.683002, 0.683002, -0.183051], [0,0,0,0], [9E9, 9E9, 9E9, 9E9, 9E9, 9E9]];
	VAR robtarget Openhole_903 := [[536.38, -35.46, 190.47], [0.183051, 0.683002, 0.683002, -0.183051], [0,0,0,0], [9E9, 9E9, 9E9, 9E9, 9E9, 9E9]];
	VAR robtarget Openhole_904 := [[509.38, -35.46, 190.55], [0.183051, 0.683002, 0.683002, -0.183051], [0,0,0,0], [9E9, 9E9, 9E9, 9E9, 9E9, 9E9]];
	VAR robtarget Openhole_905 := [[504.37, -35.46, 189.76], [0.218209, 0.672596, 0.696508, -0.121972], [0,0,0,0], [9E9, 9E9, 9E9, 9E9, 9E9, 9E9]];
	VAR robtarget Openhole_906 := [[504.37, -35.46, 189.76], [0.218204, 0.672597, 0.696509, -0.121965], [0,0,0,0], [9E9, 9E9, 9E9, 9E9, 9E9, 9E9]];
	VAR robtarget Openhole_907 := [[503.88, -35.49, 189.7], [0.217132, 0.672944, 0.696768, -0.120478], [0,0,0,0], [9E9, 9E9, 9E9, 9E9, 9E9, 9E9]];
	VAR robtarget Openhole_908 := [[492, -36.34, 188.16], [0.190087, 0.681078, 0.702238, -0.082839], [0,0,0,0], [9E9, 9E9, 9E9, 9E9, 9E9, 9E9]];
	VAR robtarget Openhole_909 := [[483.63, -37.25, 187.07], [0.170072, 0.686349, 0.705078, -0.053531], [0,0,0,0], [9E9, 9E9, 9E9, 9E9, 9E9, 9E9]];
	VAR robtarget Openhole_910 := [[476.28, -38.4, 186.08], [0.152443, 0.690479, 0.706639, -0.025703], [0,0,0,0], [9E9, 9E9, 9E9, 9E9, 9E9, 9E9]];
	VAR robtarget Openhole_911 := [[475.31, -38.59, 185.95], [0.150126, 0.690986, 0.706769, -0.021855], [0,0,0,0], [9E9, 9E9, 9E9, 9E9, 9E9, 9E9]];
	VAR robtarget Openhole_912 := [[474.82, -38.7, 185.88], [0.149025, 0.691225, 0.706828, -0.019855], [0,0,0,0], [9E9, 9E9, 9E9, 9E9, 9E9, 9E9]];
	VAR robtarget Openhole_913 := [[470.42, -38.7, 185.05], [0.135674, 0.693969, 0.707089, -0.004992], [0,0,0,0], [9E9, 9E9, 9E9, 9E9, 9E9, 9E9]];
	VAR robtarget Openhole_914 := [[470.91, -38.55, 185.11], [0.136697, 0.693768, 0.707071, -0.007116], [0,0,0,0], [9E9, 9E9, 9E9, 9E9, 9E9, 9E9]];
	VAR robtarget Openhole_915 := [[477.71, -37.2, 186.02], [0.152931, 0.690371, 0.706274, -0.034308], [0,0,0,0], [9E9, 9E9, 9E9, 9E9, 9E9, 9E9]];
	VAR robtarget Openhole_916 := [[485.08, -36.14, 186.94], [0.170773, 0.686175, 0.704411, -0.061683], [0,0,0,0], [9E9, 9E9, 9E9, 9E9, 9E9, 9E9]];
	VAR robtarget Openhole_917 := [[493.97, -35.28, 188.04], [0.192098, 0.680513, 0.701087, -0.092067], [0,0,0,0], [9E9, 9E9, 9E9, 9E9, 9E9, 9E9]];
	VAR robtarget Openhole_918 := [[504.37, -34.58, 189.29], [0.215729, 0.673395, 0.696052, -0.124544], [0,0,0,0], [9E9, 9E9, 9E9, 9E9, 9E9, 9E9]];
	VAR robtarget Openhole_919 := [[509.37, -34.58, 190.04], [0.183051, 0.683002, 0.683002, -0.183051], [0,0,0,0], [9E9, 9E9, 9E9, 9E9, 9E9, 9E9]];
	VAR robtarget Openhole_920 := [[536.37, -34.58, 189.96], [0.183051, 0.683002, 0.683002, -0.183051], [0,0,0,0], [9E9, 9E9, 9E9, 9E9, 9E9, 9E9]];
	VAR robtarget Openhole_921 := [[536.37, -33.69, 189.45], [0.183051, 0.683002, 0.683002, -0.183051], [0,0,0,0], [9E9, 9E9, 9E9, 9E9, 9E9, 9E9]];
	VAR robtarget Openhole_922 := [[524.37, -33.69, 189.48], [0.183051, 0.683002, 0.683002, -0.183051], [0,0,0,0], [9E9, 9E9, 9E9, 9E9, 9E9, 9E9]];
	VAR robtarget Openhole_923 := [[509.37, -33.69, 189.53], [0.183051, 0.683002, 0.683002, -0.183051], [0,0,0,0], [9E9, 9E9, 9E9, 9E9, 9E9, 9E9]];
	VAR robtarget Openhole_924 := [[504.38, -33.69, 188.83], [0.213252, 0.674184, 0.695584, -0.127132], [0,0,0,0], [9E9, 9E9, 9E9, 9E9, 9E9, 9E9]];
	VAR robtarget Openhole_925 := [[490, -34.71, 187.2], [0.179938, 0.683829, 0.702379, -0.081628], [0,0,0,0], [9E9, 9E9, 9E9, 9E9, 9E9, 9E9]];
	VAR robtarget Openhole_926 := [[482.1, -35.58, 186.28], [0.160641, 0.688618, 0.705053, -0.053852], [0,0,0,0], [9E9, 9E9, 9E9, 9E9, 9E9, 9E9]];
	VAR robtarget Openhole_927 := [[475.24, -36.68, 185.46], [0.143944, 0.692301, 0.706563, -0.027734], [0,0,0,0], [9E9, 9E9, 9E9, 9E9, 9E9, 9E9]];
	VAR robtarget Openhole_928 := [[467.96, -38.24, 184.5], [0.126592, 0.695683, 0.707104, 0.00189], [0,0,0,0], [9E9, 9E9, 9E9, 9E9, 9E9, 9E9]];
	VAR robtarget Openhole_929 := [[467, -38.47, 184.36], [0.124297, 0.696096, 0.707082, 0.005923], [0,0,0,0], [9E9, 9E9, 9E9, 9E9, 9E9, 9E9]];
	VAR robtarget Openhole_930 := [[466.52, -38.7, 184.31], [0.123499, 0.696238, 0.707058, 0.008325], [0,0,0,0], [9E9, 9E9, 9E9, 9E9, 9E9, 9E9]];
	VAR robtarget Openhole_931 := [[462.13, -38.7, 183.48], [0.109513, 0.698575, 0.706721, 0.023347], [0,0,0,0], [9E9, 9E9, 9E9, 9E9, 9E9, 9E9]];
	VAR robtarget Openhole_932 := [[462.62, -38.48, 183.54], [0.11035, 0.698443, 0.706796, 0.02096], [0,0,0,0], [9E9, 9E9, 9E9, 9E9, 9E9, 9E9]];
	VAR robtarget Openhole_933 := [[471.3, -36.44, 184.74], [0.131223, 0.694824, 0.706942, -0.01528], [0,0,0,0], [9E9, 9E9, 9E9, 9E9, 9E9, 9E9]];
	VAR robtarget Openhole_934 := [[478.14, -35.16, 185.53], [0.147835, 0.69148, 0.705846, -0.042213], [0,0,0,0], [9E9, 9E9, 9E9, 9E9, 9E9, 9E9]];
	VAR robtarget Openhole_935 := [[485.53, -34.21, 186.35], [0.16616, 0.687307, 0.703716, -0.069164], [0,0,0,0], [9E9, 9E9, 9E9, 9E9, 9E9, 9E9]];
	VAR robtarget Openhole_936 := [[495.44, -33.39, 187.43], [0.19032, 0.681013, 0.699679, -0.102218], [0,0,0,0], [9E9, 9E9, 9E9, 9E9, 9E9, 9E9]];
	VAR robtarget Openhole_937 := [[504.38, -32.81, 188.36], [0.210762, 0.674966, 0.695107, -0.129717], [0,0,0,0], [9E9, 9E9, 9E9, 9E9, 9E9, 9E9]];
	VAR robtarget Openhole_938 := [[509.37, -32.81, 189.02], [0.183051, 0.683002, 0.683002, -0.183051], [0,0,0,0], [9E9, 9E9, 9E9, 9E9, 9E9, 9E9]];
	VAR robtarget Openhole_939 := [[536.37, -32.81, 188.94], [0.183051, 0.683002, 0.683002, -0.183051], [0,0,0,0], [9E9, 9E9, 9E9, 9E9, 9E9, 9E9]];
	VAR robtarget Openhole_940 := [[536.37, -31.93, 188.43], [0.183051, 0.683002, 0.683002, -0.183051], [0,0,0,0], [9E9, 9E9, 9E9, 9E9, 9E9, 9E9]];
	VAR robtarget Openhole_941 := [[524.37, -31.93, 188.46], [0.183051, 0.683002, 0.683002, -0.183051], [0,0,0,0], [9E9, 9E9, 9E9, 9E9, 9E9, 9E9]];
	VAR robtarget Openhole_942 := [[509.37, -31.93, 188.51], [0.183051, 0.683002, 0.683002, -0.183051], [0,0,0,0], [9E9, 9E9, 9E9, 9E9, 9E9, 9E9]];
	VAR robtarget Openhole_943 := [[504.38, -31.93, 187.89], [0.208265, 0.675741, 0.694619, -0.132304], [0,0,0,0], [9E9, 9E9, 9E9, 9E9, 9E9, 9E9]];
	VAR robtarget Openhole_944 := [[487.98, -33.03, 186.27], [0.16938, 0.68652, 0.702499, -0.080596], [0,0,0,0], [9E9, 9E9, 9E9, 9E9, 9E9, 9E9]];
	VAR robtarget Openhole_945 := [[479.58, -33.93, 185.4], [0.148213, 0.691399, 0.705272, -0.050912], [0,0,0,0], [9E9, 9E9, 9E9, 9E9, 9E9, 9E9]];
	VAR robtarget Openhole_946 := [[473.19, -34.93, 184.71], [0.132249, 0.69463, 0.706608, -0.026547], [0,0,0,0], [9E9, 9E9, 9E9, 9E9, 9E9, 9E9]];
	VAR robtarget Openhole_947 := [[466.4, -36.39, 183.91], [0.115743, 0.69757, 0.707106, 0.001214], [0,0,0,0], [9E9, 9E9, 9E9, 9E9, 9E9, 9E9]];
	VAR robtarget Openhole_948 := [[457.75, -38.56, 182.64], [0.09478, 0.700726, 0.706089, 0.037918], [0,0,0,0], [9E9, 9E9, 9E9, 9E9, 9E9, 9E9]];
	VAR robtarget Openhole_949 := [[457.27, -38.7, 182.56], [0.093663, 0.700876, 0.705973, 0.040025], [0,0,0,0], [9E9, 9E9, 9E9, 9E9, 9E9, 9E9]];
	VAR robtarget Openhole_950 := [[452.92, -38.7, 181.74], [0.079195, 0.702658, 0.70497, 0.054933], [0,0,0,0], [9E9, 9E9, 9E9, 9E9, 9E9, 9E9]];
	VAR robtarget Openhole_951 := [[460.54, -36.57, 182.95], [0.097469, 0.700357, 0.706769, 0.021843], [0,0,0,0], [9E9, 9E9, 9E9, 9E9, 9E9, 9E9]];
	VAR robtarget Openhole_952 := [[467.77, -34.81, 183.86], [0.114999, 0.697693, 0.707054, -0.008654], [0,0,0,0], [9E9, 9E9, 9E9, 9E9, 9E9, 9E9]];
	VAR robtarget Openhole_953 := [[474.13, -33.64, 184.55], [0.130984, 0.694869, 0.706295, -0.033864], [0,0,0,0], [9E9, 9E9, 9E9, 9E9, 9E9, 9E9]];
	VAR robtarget Openhole_954 := [[481.53, -32.67, 185.28], [0.149966, 0.691021, 0.704448, -0.061258], [0,0,0,0], [9E9, 9E9, 9E9, 9E9, 9E9, 9E9]];
	VAR robtarget Openhole_955 := [[491.44, -31.83, 186.25], [0.175168, 0.685067, 0.700699, -0.09498], [0,0,0,0], [9E9, 9E9, 9E9, 9E9, 9E9, 9E9]];
	VAR robtarget Openhole_956 := [[504.38, -31.04, 187.42], [0.205767, 0.676506, 0.694119, -0.134901], [0,0,0,0], [9E9, 9E9, 9E9, 9E9, 9E9, 9E9]];
	VAR robtarget Openhole_957 := [[509.37, -31.04, 188], [0.183051, 0.683002, 0.683002, -0.183051], [0,0,0,0], [9E9, 9E9, 9E9, 9E9, 9E9, 9E9]];
	VAR robtarget Openhole_958 := [[536.33, -31.04, 187.92], [0.183051, 0.683002, 0.683002, -0.183051], [0,0,0,0], [9E9, 9E9, 9E9, 9E9, 9E9, 9E9]];
	VAR robtarget Openhole_959 := [[536.24, -21.49, 182.4], [0.183051, 0.683002, 0.683002, -0.183051], [0,0,0,0], [9E9, 9E9, 9E9, 9E9, 9E9, 9E9]];
	VAR robtarget Openhole_960 := [[509.35, -21.49, 182.49], [0.183051, 0.683002, 0.683002, -0.183051], [0,0,0,0], [9E9, 9E9, 9E9, 9E9, 9E9, 9E9]];
	VAR robtarget Openhole_961 := [[504.35, -21.49, 182.37], [0.178251, 0.684271, 0.688104, -0.162827], [0,0,0,0], [9E9, 9E9, 9E9, 9E9, 9E9, 9E9]];
	VAR robtarget Openhole_962 := [[503.38, -21.52, 182.36], [0.175882, 0.684884, 0.688724, -0.160183], [0,0,0,0], [9E9, 9E9, 9E9, 9E9, 9E9, 9E9]];
	VAR robtarget Openhole_963 := [[493.89, -21.85, 182.27], [0.151582, 0.690668, 0.694477, -0.133047], [0,0,0,0], [9E9, 9E9, 9E9, 9E9, 9E9, 9E9]];
	VAR robtarget Openhole_964 := [[487.39, -21.9, 182.11], [0.133303, 0.694428, 0.697884, -0.113832], [0,0,0,0], [9E9, 9E9, 9E9, 9E9, 9E9, 9E9]];
	VAR robtarget Openhole_965 := [[486.89, -21.89, 182.1], [0.131846, 0.694706, 0.698127, -0.112332], [0,0,0,0], [9E9, 9E9, 9E9, 9E9, 9E9, 9E9]];
	VAR robtarget Openhole_966 := [[473.4, -21.68, 181.68], [0.090004, 0.701355, 0.703557, -0.070759], [0,0,0,0], [9E9, 9E9, 9E9, 9E9, 9E9, 9E9]];
	VAR robtarget Openhole_967 := [[465.91, -21.31, 181.43], [0.064606, 0.704149, 0.705519, -0.047355], [0,0,0,0], [9E9, 9E9, 9E9, 9E9, 9E9, 9E9]];
	VAR robtarget Openhole_968 := [[463.92, -21.12, 181.36], [0.057418, 0.704772, 0.705897, -0.041343], [0,0,0,0], [9E9, 9E9, 9E9, 9E9, 9E9, 9E9]];
	VAR robtarget Openhole_969 := [[457.02, -21.12, 181.22], [0.034362, 0.706271, 0.706877, -0.018031], [0,0,0,0], [9E9, 9E9, 9E9, 9E9, 9E9, 9E9]];
	VAR robtarget Openhole_970 := [[456.81, -15.81, 180.83], [0.015661, 0.706933, 0.706222, -0.035353], [0,0,0,0], [9E9, 9E9, 9E9, 9E9, 9E9, 9E9]];
	VAR robtarget Openhole_971 := [[457.68, -15.38, 180.77], [0.01717, 0.706898, 0.705987, -0.03978], [0,0,0,0], [9E9, 9E9, 9E9, 9E9, 9E9, 9E9]];
	VAR robtarget Openhole_972 := [[458.51, -14.82, 180.69], [0.018053, 0.706876, 0.705708, -0.044459], [0,0,0,0], [9E9, 9E9, 9E9, 9E9, 9E9, 9E9]];
	VAR robtarget Openhole_973 := [[460.62, -13.5, 180.46], [0.020761, 0.706802, 0.704887, -0.05599], [0,0,0,0], [9E9, 9E9, 9E9, 9E9, 9E9, 9E9]];
	VAR robtarget Openhole_974 := [[461.06, -13.27, 180.41], [0.021468, 0.706781, 0.704704, -0.058241], [0,0,0,0], [9E9, 9E9, 9E9, 9E9, 9E9, 9E9]];
	VAR robtarget Openhole_975 := [[460.89, -17, 180.84], [0.03344, 0.706316, 0.705669, -0.045077], [0,0,0,0], [9E9, 9E9, 9E9, 9E9, 9E9, 9E9]];
	VAR robtarget Openhole_976 := [[462.52, -15.87, 180.66], [0.0351, 0.706235, 0.705012, -0.054389], [0,0,0,0], [9E9, 9E9, 9E9, 9E9, 9E9, 9E9]];
	VAR robtarget Openhole_977 := [[462.94, -15.6, 180.61], [0.035601, 0.70621, 0.704831, -0.056691], [0,0,0,0], [9E9, 9E9, 9E9, 9E9, 9E9, 9E9]];
	VAR robtarget Openhole_978 := [[463.79, -15.08, 180.51], [0.036721, 0.706153, 0.704449, -0.061252], [0,0,0,0], [9E9, 9E9, 9E9, 9E9, 9E9, 9E9]];
	VAR robtarget Openhole_979 := [[464.66, -14.6, 180.41], [0.037997, 0.706085, 0.704043, -0.065755], [0,0,0,0], [9E9, 9E9, 9E9, 9E9, 9E9, 9E9]];
	VAR robtarget Openhole_980 := [[465.55, -14.15, 180.3], [0.039457, 0.706005, 0.703615, -0.070183], [0,0,0,0], [9E9, 9E9, 9E9, 9E9, 9E9, 9E9]];
	VAR robtarget Openhole_981 := [[466, -13.94, 180.25], [0.040259, 0.70596, 0.703394, -0.072365], [0,0,0,0], [9E9, 9E9, 9E9, 9E9, 9E9, 9E9]];
	VAR robtarget Openhole_982 := [[466.46, -13.74, 180.19], [0.041104, 0.705911, 0.703169, -0.074525], [0,0,0,0], [9E9, 9E9, 9E9, 9E9, 9E9, 9E9]];
	VAR robtarget Openhole_983 := [[467.38, -13.37, 180.08], [0.042935, 0.705802, 0.702705, -0.078774], [0,0,0,0], [9E9, 9E9, 9E9, 9E9, 9E9, 9E9]];
	VAR robtarget Openhole_984 := [[467.84, -13.2, 180.02], [0.043911, 0.705742, 0.702468, -0.080865], [0,0,0,0], [9E9, 9E9, 9E9, 9E9, 9E9, 9E9]];
	VAR robtarget Openhole_985 := [[468.32, -13.04, 179.97], [0.044946, 0.705677, 0.702228, -0.082921], [0,0,0,0], [9E9, 9E9, 9E9, 9E9, 9E9, 9E9]];
	VAR robtarget Openhole_986 := [[469.27, -12.75, 179.86], [0.047121, 0.705535, 0.701739, -0.086964], [0,0,0,0], [9E9, 9E9, 9E9, 9E9, 9E9, 9E9]];
	VAR robtarget Openhole_987 := [[470.71, -12.36, 179.69], [0.050581, 0.705295, 0.700981, -0.092878], [0,0,0,0], [9E9, 9E9, 9E9, 9E9, 9E9, 9E9]];
	VAR robtarget Openhole_988 := [[471.19, -12.25, 179.64], [0.051803, 0.705207, 0.700724, -0.094796], [0,0,0,0], [9E9, 9E9, 9E9, 9E9, 9E9, 9E9]];
	VAR robtarget Openhole_989 := [[471.68, -12.15, 179.58], [0.053062, 0.705113, 0.700466, -0.096685], [0,0,0,0], [9E9, 9E9, 9E9, 9E9, 9E9, 9E9]];
	VAR robtarget Openhole_990 := [[475.61, -11.57, 179.18], [0.063959, 0.704208, 0.698342, -0.11099], [0,0,0,0], [9E9, 9E9, 9E9, 9E9, 9E9, 9E9]];
	VAR robtarget Openhole_991 := [[480.08, -11.3, 178.78], [0.077398, 0.702858, 0.695866, -0.125581], [0,0,0,0], [9E9, 9E9, 9E9, 9E9, 9E9, 9E9]];
	VAR robtarget Openhole_992 := [[482.58, -11.27, 178.58], [0.085139, 0.701963, 0.694457, -0.133149], [0,0,0,0], [9E9, 9E9, 9E9, 9E9, 9E9, 9E9]];
	VAR robtarget Openhole_993 := [[483.08, -11.27, 178.54], [0.086697, 0.701772, 0.694173, -0.134626], [0,0,0,0], [9E9, 9E9, 9E9, 9E9, 9E9, 9E9]];
	VAR robtarget Openhole_994 := [[497.54, -11.57, 177.6], [0.130615, 0.694939, 0.685287, -0.174302], [0,0,0,0], [9E9, 9E9, 9E9, 9E9, 9E9, 9E9]];
	VAR robtarget Openhole_995 := [[498.04, -11.57, 177.56], [0.132014, 0.694674, 0.68495, -0.175623], [0,0,0,0], [9E9, 9E9, 9E9, 9E9, 9E9, 9E9]];
	VAR robtarget Openhole_996 := [[503.02, -11.41, 177.12], [0.145263, 0.692025, 0.68141, -0.188892], [0,0,0,0], [9E9, 9E9, 9E9, 9E9, 9E9, 9E9]];
	VAR robtarget Openhole_997 := [[503.51, -11.37, 177.07], [0.14651, 0.691762, 0.681039, -0.190227], [0,0,0,0], [9E9, 9E9, 9E9, 9E9, 9E9, 9E9]];
	VAR robtarget Openhole_998 := [[504.33, -11.35, 177], [0.148641, 0.691307, 0.680445, -0.192339], [0,0,0,0], [9E9, 9E9, 9E9, 9E9, 9E9, 9E9]];
	VAR robtarget Openhole_999 := [[509.33, -11.35, 176.63], [0.183051, 0.683002, 0.683002, -0.183051], [0,0,0,0], [9E9, 9E9, 9E9, 9E9, 9E9, 9E9]];
	VAR robtarget Openhole_1000 := [[536.33, -11.35, 176.54], [0.183051, 0.683002, 0.683002, -0.183051], [0,0,0,0], [9E9, 9E9, 9E9, 9E9, 9E9, 9E9]];
	VAR robtarget Openhole_1001 := [[536.34, -13.35, 177.7], [0.183051, 0.683002, 0.683002, -0.183051], [0,0,0,0], [9E9, 9E9, 9E9, 9E9, 9E9, 9E9]];
	VAR robtarget Openhole_1002 := [[509.34, -13.35, 177.78], [0.183051, 0.683002, 0.683002, -0.183051], [0,0,0,0], [9E9, 9E9, 9E9, 9E9, 9E9, 9E9]];
	VAR robtarget Openhole_1003 := [[504.34, -13.35, 178.05], [0.154483, 0.690025, 0.682051, -0.186566], [0,0,0,0], [9E9, 9E9, 9E9, 9E9, 9E9, 9E9]];
	VAR robtarget Openhole_1004 := [[498.25, -13.65, 178.53], [0.13886, 0.693338, 0.686377, -0.16996], [0,0,0,0], [9E9, 9E9, 9E9, 9E9, 9E9, 9E9]];
	VAR robtarget Openhole_1005 := [[494.75, -13.69, 178.73], [0.129132, 0.695216, 0.688667, -0.160428], [0,0,0,0], [9E9, 9E9, 9E9, 9E9, 9E9, 9E9]];
	VAR robtarget Openhole_1006 := [[494.26, -13.69, 178.75], [0.127703, 0.69548, 0.688985, -0.15906], [0,0,0,0], [9E9, 9E9, 9E9, 9E9, 9E9, 9E9]];
	VAR robtarget Openhole_1007 := [[482.27, -13.53, 179.32], [0.091393, 0.701176, 0.695961, -0.125056], [0,0,0,0], [9E9, 9E9, 9E9, 9E9, 9E9, 9E9]];
	VAR robtarget Openhole_1008 := [[481.77, -13.53, 179.35], [0.089843, 0.701376, 0.696229, -0.123551], [0,0,0,0], [9E9, 9E9, 9E9, 9E9, 9E9, 9E9]];
	VAR robtarget Openhole_1009 := [[476.28, -13.68, 179.67], [0.073003, 0.703328, 0.699083, -0.106221], [0,0,0,0], [9E9, 9E9, 9E9, 9E9, 9E9, 9E9]];
	VAR robtarget Openhole_1010 := [[474.29, -13.82, 179.81], [0.067076, 0.703918, 0.700071, -0.0995], [0,0,0,0], [9E9, 9E9, 9E9, 9E9, 9E9, 9E9]];
	VAR robtarget Openhole_1011 := [[473.3, -13.93, 179.89], [0.064232, 0.704183, 0.70056, -0.095999], [0,0,0,0], [9E9, 9E9, 9E9, 9E9, 9E9, 9E9]];
	VAR robtarget Openhole_1012 := [[470.85, -19.93, 181.25], [0.07609, 0.703001, 0.703802, -0.068286], [0,0,0,0], [9E9, 9E9, 9E9, 9E9, 9E9, 9E9]];
	VAR robtarget Openhole_1013 := [[487.35, -20.27, 181.51], [0.128076, 0.695411, 0.697047, -0.118853], [0,0,0,0], [9E9, 9E9, 9E9, 9E9, 9E9, 9E9]];
	VAR robtarget Openhole_1014 := [[489.35, -20.27, 181.54], [0.133906, 0.694312, 0.696014, -0.124758], [0,0,0,0], [9E9, 9E9, 9E9, 9E9, 9E9, 9E9]];
	VAR robtarget Openhole_1015 := [[489.85, -20.27, 181.55], [0.135344, 0.694033, 0.695749, -0.126227], [0,0,0,0], [9E9, 9E9, 9E9, 9E9, 9E9, 9E9]];
	VAR robtarget Openhole_1016 := [[499.85, -20.1, 181.58], [0.162464, 0.68819, 0.689918, -0.15496], [0,0,0,0], [9E9, 9E9, 9E9, 9E9, 9E9, 9E9]];
	VAR robtarget Openhole_1017 := [[504.35, -19.88, 181.52], [0.173568, 0.685474, 0.686973, -0.167536], [0,0,0,0], [9E9, 9E9, 9E9, 9E9, 9E9, 9E9]];
	VAR robtarget Openhole_1018 := [[536.35, -19.88, 181.47], [0.183051, 0.683002, 0.683002, -0.183051], [0,0,0,0], [9E9, 9E9, 9E9, 9E9, 9E9, 9E9]];
	VAR robtarget Openhole_1019 := [[536.35, -19.19, 181.07], [0.183051, 0.683002, 0.683002, -0.183051], [0,0,0,0], [9E9, 9E9, 9E9, 9E9, 9E9, 9E9]];
	VAR robtarget Openhole_1020 := [[509.35, -19.19, 181.15], [0.183051, 0.683002, 0.683002, -0.183051], [0,0,0,0], [9E9, 9E9, 9E9, 9E9, 9E9, 9E9]];
	VAR robtarget Openhole_1021 := [[504.35, -19.19, 181.15], [0.171537, 0.685985, 0.686473, -0.169574], [0,0,0,0], [9E9, 9E9, 9E9, 9E9, 9E9, 9E9]];
	VAR robtarget Openhole_1022 := [[495.63, -19.51, 181.28], [0.149284, 0.691169, 0.692052, -0.145133], [0,0,0,0], [9E9, 9E9, 9E9, 9E9, 9E9, 9E9]];
	VAR robtarget Openhole_1023 := [[490.13, -19.56, 181.27], [0.133935, 0.694306, 0.695189, -0.129278], [0,0,0,0], [9E9, 9E9, 9E9, 9E9, 9E9, 9E9]];
	VAR robtarget Openhole_1024 := [[489.63, -19.56, 181.27], [0.132492, 0.694583, 0.695458, -0.127819], [0,0,0,0], [9E9, 9E9, 9E9, 9E9, 9E9, 9E9]];
	VAR robtarget Openhole_1025 := [[470.13, -19.24, 181.1], [0.071474, 0.703485, 0.703808, -0.068222], [0,0,0,0], [9E9, 9E9, 9E9, 9E9, 9E9, 9E9]];
	VAR robtarget Openhole_1026 := [[469.63, -19.24, 181.1], [0.069853, 0.703648, 0.703965, -0.066584], [0,0,0,0], [9E9, 9E9, 9E9, 9E9, 9E9, 9E9]];
	VAR robtarget Openhole_1027 := [[469.13, -19.24, 181.1], [0.068219, 0.703808, 0.704117, -0.064953], [0,0,0,0], [9E9, 9E9, 9E9, 9E9, 9E9, 9E9]];
	VAR robtarget Openhole_1028 := [[466.63, -19.31, 181.11], [0.060282, 0.704533, 0.704848, -0.056474], [0,0,0,0], [9E9, 9E9, 9E9, 9E9, 9E9, 9E9]];
	VAR robtarget Openhole_1029 := [[466.13, -19.31, 181.11], [0.05865, 0.70467, 0.70498, -0.054803], [0,0,0,0], [9E9, 9E9, 9E9, 9E9, 9E9, 9E9]];
	VAR robtarget Openhole_1030 := [[465.63, -19.33, 181.11], [0.057055, 0.704801, 0.705111, -0.053092], [0,0,0,0], [9E9, 9E9, 9E9, 9E9, 9E9, 9E9]];
	VAR robtarget Openhole_1031 := [[464.64, -19.38, 181.11], [0.053941, 0.705046, 0.705366, -0.049583], [0,0,0,0], [9E9, 9E9, 9E9, 9E9, 9E9, 9E9]];
	VAR robtarget Openhole_1032 := [[464.14, -19.42, 181.12], [0.052423, 0.705161, 0.70549, -0.047787], [0,0,0,0], [9E9, 9E9, 9E9, 9E9, 9E9, 9E9]];
	VAR robtarget Openhole_1033 := [[463.64, -19.43, 181.12], [0.050789, 0.70528, 0.705603, -0.046092], [0,0,0,0], [9E9, 9E9, 9E9, 9E9, 9E9, 9E9]];
	VAR robtarget Openhole_1034 := [[462.64, -19.54, 181.13], [0.047837, 0.705487, 0.705834, -0.042407], [0,0,0,0], [9E9, 9E9, 9E9, 9E9, 9E9, 9E9]];
	VAR robtarget Openhole_1035 := [[462.14, -19.58, 181.13], [0.046317, 0.705588, 0.705941, -0.040595], [0,0,0,0], [9E9, 9E9, 9E9, 9E9, 9E9, 9E9]];
	VAR robtarget Openhole_1036 := [[461.97, -18.21, 180.96], [0.041126, 0.70591, 0.705697, -0.044632], [0,0,0,0], [9E9, 9E9, 9E9, 9E9, 9E9, 9E9]];
	VAR robtarget Openhole_1037 := [[462.42, -18, 180.93], [0.041929, 0.705863, 0.705552, -0.046858], [0,0,0,0], [9E9, 9E9, 9E9, 9E9, 9E9, 9E9]];
	VAR robtarget Openhole_1038 := [[462.86, -17.76, 180.9], [0.042609, 0.705822, 0.705398, -0.049122], [0,0,0,0], [9E9, 9E9, 9E9, 9E9, 9E9, 9E9]];
	VAR robtarget Openhole_1039 := [[463.78, -17.37, 180.83], [0.044369, 0.705713, 0.70508, -0.053498], [0,0,0,0], [9E9, 9E9, 9E9, 9E9, 9E9, 9E9]];
	VAR robtarget Openhole_1040 := [[465.15, -16.77, 180.72], [0.046875, 0.705551, 0.70455, -0.060082], [0,0,0,0], [9E9, 9E9, 9E9, 9E9, 9E9, 9E9]];
	VAR robtarget Openhole_1041 := [[465.61, -16.58, 180.68], [0.047764, 0.705492, 0.704362, -0.062245], [0,0,0,0], [9E9, 9E9, 9E9, 9E9, 9E9, 9E9]];
	VAR robtarget Openhole_1042 := [[466.54, -16.21, 180.6], [0.049629, 0.705363, 0.703971, -0.066523], [0,0,0,0], [9E9, 9E9, 9E9, 9E9, 9E9, 9E9]];
	VAR robtarget Openhole_1043 := [[467.01, -16.05, 180.56], [0.05063, 0.705292, 0.703769, -0.068623], [0,0,0,0], [9E9, 9E9, 9E9, 9E9, 9E9, 9E9]];
	VAR robtarget Openhole_1044 := [[468.44, -15.62, 180.44], [0.053935, 0.705047, 0.703146, -0.07474], [0,0,0,0], [9E9, 9E9, 9E9, 9E9, 9E9, 9E9]];
	VAR robtarget Openhole_1045 := [[469.4, -15.37, 180.36], [0.056272, 0.704864, 0.702712, -0.078716], [0,0,0,0], [9E9, 9E9, 9E9, 9E9, 9E9, 9E9]];
	VAR robtarget Openhole_1046 := [[471.36, -14.97, 180.2], [0.061337, 0.704441, 0.701814, -0.086357], [0,0,0,0], [9E9, 9E9, 9E9, 9E9, 9E9, 9E9]];
	VAR robtarget Openhole_1047 := [[471.85, -14.89, 180.17], [0.062673, 0.704324, 0.701584, -0.088205], [0,0,0,0], [9E9, 9E9, 9E9, 9E9, 9E9, 9E9]];
	VAR robtarget Openhole_1048 := [[472.34, -14.82, 180.13], [0.064046, 0.7042, 0.701353, -0.090019], [0,0,0,0], [9E9, 9E9, 9E9, 9E9, 9E9, 9E9]];
	VAR robtarget Openhole_1049 := [[476.32, -14.47, 179.88], [0.075703, 0.703043, 0.699454, -0.10375], [0,0,0,0], [9E9, 9E9, 9E9, 9E9, 9E9, 9E9]];
	VAR robtarget Openhole_1050 := [[480.81, -14.37, 179.65], [0.089568, 0.701411, 0.697202, -0.11794], [0,0,0,0], [9E9, 9E9, 9E9, 9E9, 9E9, 9E9]];
	VAR robtarget Openhole_1051 := [[481.31, -14.37, 179.63], [0.091126, 0.70121, 0.696944, -0.119456], [0,0,0,0], [9E9, 9E9, 9E9, 9E9, 9E9, 9E9]];
	VAR robtarget Openhole_1052 := [[493.8, -14.52, 179.13], [0.128934, 0.695252, 0.689846, -0.155283], [0,0,0,0], [9E9, 9E9, 9E9, 9E9, 9E9, 9E9]];
	VAR robtarget Openhole_1053 := [[494.3, -14.52, 179.11], [0.130362, 0.694986, 0.689534, -0.156663], [0,0,0,0], [9E9, 9E9, 9E9, 9E9, 9E9, 9E9]];
	VAR robtarget Openhole_1054 := [[501.29, -14.35, 178.72], [0.149266, 0.691173, 0.684889, -0.175862], [0,0,0,0], [9E9, 9E9, 9E9, 9E9, 9E9, 9E9]];
	VAR robtarget Openhole_1055 := [[504.34, -14.15, 178.48], [0.156823, 0.689497, 0.682681, -0.184247], [0,0,0,0], [9E9, 9E9, 9E9, 9E9, 9E9, 9E9]];
	VAR robtarget Openhole_1056 := [[509.34, -14.15, 178.24], [0.183051, 0.683002, 0.683002, -0.183051], [0,0,0,0], [9E9, 9E9, 9E9, 9E9, 9E9, 9E9]];
	VAR robtarget Openhole_1057 := [[536.34, -14.15, 178.16], [0.183051, 0.683002, 0.683002, -0.183051], [0,0,0,0], [9E9, 9E9, 9E9, 9E9, 9E9, 9E9]];
	VAR robtarget Openhole_1058 := [[536.34, -15.36, 178.86], [0.183051, 0.683002, 0.683002, -0.183051], [0,0,0,0], [9E9, 9E9, 9E9, 9E9, 9E9, 9E9]];
	VAR robtarget Openhole_1059 := [[509.34, -15.36, 178.94], [0.183051, 0.683002, 0.683002, -0.183051], [0,0,0,0], [9E9, 9E9, 9E9, 9E9, 9E9, 9E9]];
	VAR robtarget Openhole_1060 := [[504.34, -15.36, 179.12], [0.160357, 0.688684, 0.683618, -0.180737], [0,0,0,0], [9E9, 9E9, 9E9, 9E9, 9E9, 9E9]];
	VAR robtarget Openhole_1061 := [[503.64, -15.39, 179.16], [0.158619, 0.689086, 0.684109, -0.178871], [0,0,0,0], [9E9, 9E9, 9E9, 9E9, 9E9, 9E9]];
	VAR robtarget Openhole_1062 := [[497.66, -15.67, 179.5], [0.143301, 0.692434, 0.688222, -0.16233], [0,0,0,0], [9E9, 9E9, 9E9, 9E9, 9E9, 9E9]];
	VAR robtarget Openhole_1063 := [[492.66, -15.73, 179.69], [0.1294, 0.695166, 0.691361, -0.14839], [0,0,0,0], [9E9, 9E9, 9E9, 9E9, 9E9, 9E9]];
	VAR robtarget Openhole_1064 := [[492.16, -15.73, 179.7], [0.12796, 0.695432, 0.691661, -0.146985], [0,0,0,0], [9E9, 9E9, 9E9, 9E9, 9E9, 9E9]];
	VAR robtarget Openhole_1065 := [[479.17, -15.58, 180.07], [0.088333, 0.701568, 0.698654, -0.109007], [0,0,0,0], [9E9, 9E9, 9E9, 9E9, 9E9, 9E9]];
	VAR robtarget Openhole_1066 := [[478.67, -15.58, 180.09], [0.086767, 0.701763, 0.698894, -0.107458], [0,0,0,0], [9E9, 9E9, 9E9, 9E9, 9E9, 9E9]];
	VAR robtarget Openhole_1067 := [[473.18, -15.79, 180.32], [0.069942, 0.703639, 0.70142, -0.089502], [0,0,0,0], [9E9, 9E9, 9E9, 9E9, 9E9, 9E9]];
	VAR robtarget Openhole_1068 := [[472.19, -15.88, 180.37], [0.067012, 0.703924, 0.701854, -0.086027], [0,0,0,0], [9E9, 9E9, 9E9, 9E9, 9E9, 9E9]];
	VAR robtarget Openhole_1069 := [[470.21, -16.14, 180.48], [0.06143, 0.704433, 0.702705, -0.078777], [0,0,0,0], [9E9, 9E9, 9E9, 9E9, 9E9, 9E9]];
	VAR robtarget Openhole_1070 := [[469.71, -16.22, 180.51], [0.06011, 0.704547, 0.702913, -0.076894], [0,0,0,0], [9E9, 9E9, 9E9, 9E9, 9E9, 9E9]];
	VAR robtarget Openhole_1071 := [[469.22, -16.32, 180.54], [0.058826, 0.704656, 0.70312, -0.07498], [0,0,0,0], [9E9, 9E9, 9E9, 9E9, 9E9, 9E9]];
	VAR robtarget Openhole_1072 := [[468.25, -16.53, 180.61], [0.056334, 0.704859, 0.703524, -0.071087], [0,0,0,0], [9E9, 9E9, 9E9, 9E9, 9E9, 9E9]];
	VAR robtarget Openhole_1073 := [[467.28, -16.77, 180.67], [0.053932, 0.705047, 0.703914, -0.067116], [0,0,0,0], [9E9, 9E9, 9E9, 9E9, 9E9, 9E9]];
	VAR robtarget Openhole_1074 := [[466.6, -18.47, 180.97], [0.057379, 0.704775, 0.704627, -0.059163], [0,0,0,0], [9E9, 9E9, 9E9, 9E9, 9E9, 9E9]];
	VAR robtarget Openhole_1075 := [[467.1, -18.42, 180.96], [0.058823, 0.704656, 0.704471, -0.060995], [0,0,0,0], [9E9, 9E9, 9E9, 9E9, 9E9, 9E9]];
	VAR robtarget Openhole_1076 := [[469.59, -18.24, 180.91], [0.066382, 0.703984, 0.703655, -0.069785], [0,0,0,0], [9E9, 9E9, 9E9, 9E9, 9E9, 9E9]];
	VAR robtarget Openhole_1077 := [[471.09, -18.16, 180.88], [0.070991, 0.703534, 0.703127, -0.07492], [0,0,0,0], [9E9, 9E9, 9E9, 9E9, 9E9, 9E9]];
	VAR robtarget Openhole_1078 := [[474.59, -18.11, 180.84], [0.082073, 0.702328, 0.701815, -0.08635], [0,0,0,0], [9E9, 9E9, 9E9, 9E9, 9E9, 9E9]];
	VAR robtarget Openhole_1079 := [[475.09, -18.11, 180.83], [0.083672, 0.702139, 0.701617, -0.087937], [0,0,0,0], [9E9, 9E9, 9E9, 9E9, 9E9, 9E9]];
	VAR robtarget Openhole_1080 := [[491.08, -18.34, 180.79], [0.132912, 0.694503, 0.693937, -0.135834], [0,0,0,0], [9E9, 9E9, 9E9, 9E9, 9E9, 9E9]];
	VAR robtarget Openhole_1081 := [[491.58, -18.34, 180.78], [0.134345, 0.694227, 0.693655, -0.137271], [0,0,0,0], [9E9, 9E9, 9E9, 9E9, 9E9, 9E9]];
	VAR robtarget Openhole_1082 := [[500.08, -18.17, 180.64], [0.157369, 0.689373, 0.688454, -0.161343], [0,0,0,0], [9E9, 9E9, 9E9, 9E9, 9E9, 9E9]];
	VAR robtarget Openhole_1083 := [[504.34, -17.96, 180.5], [0.167968, 0.686867, 0.68558, -0.173148], [0,0,0,0], [9E9, 9E9, 9E9, 9E9, 9E9, 9E9]];
	VAR robtarget Openhole_1084 := [[536.34, -17.96, 180.36], [0.183051, 0.683002, 0.683002, -0.183051], [0,0,0,0], [9E9, 9E9, 9E9, 9E9, 9E9, 9E9]];
	VAR robtarget Openhole_1085 := [[536.34, -17.24, 179.94], [0.183051, 0.683002, 0.683002, -0.183051], [0,0,0,0], [9E9, 9E9, 9E9, 9E9, 9E9, 9E9]];
	VAR robtarget Openhole_1086 := [[509.34, -17.24, 180.03], [0.183051, 0.683002, 0.683002, -0.183051], [0,0,0,0], [9E9, 9E9, 9E9, 9E9, 9E9, 9E9]];
	VAR robtarget Openhole_1087 := [[504.34, -17.24, 180.12], [0.165861, 0.687379, 0.685045, -0.175253], [0,0,0,0], [9E9, 9E9, 9E9, 9E9, 9E9, 9E9]];
	VAR robtarget Openhole_1088 := [[503.53, -17.27, 180.15], [0.163837, 0.687864, 0.685599, -0.173072], [0,0,0,0], [9E9, 9E9, 9E9, 9E9, 9E9, 9E9]];
	VAR robtarget Openhole_1089 := [[496.04, -17.57, 180.41], [0.144556, 0.692173, 0.690538, -0.152175], [0,0,0,0], [9E9, 9E9, 9E9, 9E9, 9E9, 9E9]];
	VAR robtarget Openhole_1090 := [[491.04, -17.63, 180.5], [0.130584, 0.694945, 0.693523, -0.137932], [0,0,0,0], [9E9, 9E9, 9E9, 9E9, 9E9, 9E9]];
	VAR robtarget Openhole_1091 := [[490.54, -17.62, 180.51], [0.129139, 0.695214, 0.693808, -0.136495], [0,0,0,0], [9E9, 9E9, 9E9, 9E9, 9E9, 9E9]];
	VAR robtarget Openhole_1092 := [[481.54, -17.51, 180.59], [0.1019, 0.699726, 0.698482, -0.110102], [0,0,0,0], [9E9, 9E9, 9E9, 9E9, 9E9, 9E9]];
	VAR robtarget Openhole_1093 := [[483.56, -27.51, 183.86], [0.139763, 0.693157, 0.702075, -0.084206], [0,0,0,0], [9E9, 9E9, 9E9, 9E9, 9E9, 9E9]];
	VAR robtarget Openhole_1094 := [[469.62, -28.25, 182.86], [0.099501, 0.700071, 0.706162, -0.036548], [0,0,0,0], [9E9, 9E9, 9E9, 9E9, 9E9, 9E9]];
	VAR robtarget Openhole_1095 := [[459.18, -29.01, 182.01], [0.068075, 0.703822, 0.707106, 0.001294], [0,0,0,0], [9E9, 9E9, 9E9, 9E9, 9E9, 9E9]];
	VAR robtarget Openhole_1096 := [[458.68, -29.06, 181.96], [0.066597, 0.703964, 0.7071, 0.003154], [0,0,0,0], [9E9, 9E9, 9E9, 9E9, 9E9, 9E9]];
	VAR robtarget Openhole_1097 := [[453.24, -29.67, 181.46], [0.050415, 0.705307, 0.706706, 0.02379], [0,0,0,0], [9E9, 9E9, 9E9, 9E9, 9E9, 9E9]];
	VAR robtarget Openhole_1098 := [[451.75, -29.75, 181.31], [0.045654, 0.705631, 0.706506, 0.029146], [0,0,0,0], [9E9, 9E9, 9E9, 9E9, 9E9, 9E9]];
	VAR robtarget Openhole_1099 := [[451.25, -29.75, 181.26], [0.043984, 0.705737, 0.706433, 0.030852], [0,0,0,0], [9E9, 9E9, 9E9, 9E9, 9E9, 9E9]];
	VAR robtarget Openhole_1100 := [[450.76, -29.75, 181.21], [0.042299, 0.705841, 0.706357, 0.032546], [0,0,0,0], [9E9, 9E9, 9E9, 9E9, 9E9, 9E9]];
	VAR robtarget Openhole_1101 := [[443.3, -29.47, 180.45], [0.016021, 0.706925, 0.704816, 0.056872], [0,0,0,0], [9E9, 9E9, 9E9, 9E9, 9E9, 9E9]];
	VAR robtarget Openhole_1102 := [[441.81, -29.49, 180.3], [0.011017, 0.707021, 0.704387, 0.061957], [0,0,0,0], [9E9, 9E9, 9E9, 9E9, 9E9, 9E9]];
	VAR robtarget Openhole_1103 := [[439.82, -29.61, 180.09], [0.004652, 0.707091, 0.703734, 0.06898], [0,0,0,0], [9E9, 9E9, 9E9, 9E9, 9E9, 9E9]];
	VAR robtarget Openhole_1104 := [[437.85, -29.84, 179.87], [-0.001275, 0.707106, 0.702977, 0.076306], [0,0,0,0], [9E9, 9E9, 9E9, 9E9, 9E9, 9E9]];
	VAR robtarget Openhole_1105 := [[428.05, -31.34, 178.54], [-0.029334, 0.706498, 0.698034, 0.112907], [0,0,0,0], [9E9, 9E9, 9E9, 9E9, 9E9, 9E9]];
	VAR robtarget Openhole_1106 := [[431.47, -29.27, 179.3], [-0.024708, 0.706675, 0.700663, 0.095242], [0,0,0,0], [9E9, 9E9, 9E9, 9E9, 9E9, 9E9]];
	VAR robtarget Openhole_1107 := [[437.75, -27.77, 180.09], [-0.008523, 0.707055, 0.703659, 0.069747], [0,0,0,0], [9E9, 9E9, 9E9, 9E9, 9E9, 9E9]];
	VAR robtarget Openhole_1108 := [[441.62, -26.84, 180.48], [0.001466, 0.707105, 0.705065, 0.053691], [0,0,0,0], [9E9, 9E9, 9E9, 9E9, 9E9, 9E9]];
	VAR robtarget Openhole_1109 := [[442.1, -26.73, 180.52], [0.002754, 0.707101, 0.705215, 0.051692], [0,0,0,0], [9E9, 9E9, 9E9, 9E9, 9E9, 9E9]];
	VAR robtarget Openhole_1110 := [[443.06, -26.45, 180.61], [0.005064, 0.707089, 0.705508, 0.04753], [0,0,0,0], [9E9, 9E9, 9E9, 9E9, 9E9, 9E9]];
	VAR robtarget Openhole_1111 := [[443.53, -26.29, 180.65], [0.006145, 0.70708, 0.705647, 0.045407], [0,0,0,0], [9E9, 9E9, 9E9, 9E9, 9E9, 9E9]];
	VAR robtarget Openhole_1112 := [[444.45, -25.91, 180.74], [0.007991, 0.707062, 0.705917, 0.041007], [0,0,0,0], [9E9, 9E9, 9E9, 9E9, 9E9, 9E9]];
	VAR robtarget Openhole_1113 := [[445.06, -25.46, 180.8], [0.008521, 0.707055, 0.706117, 0.037402], [0,0,0,0], [9E9, 9E9, 9E9, 9E9, 9E9, 9E9]];
	VAR robtarget Openhole_1114 := [[442.67, -23.11, 180.8], [-0.007559, 0.707066, 0.70611, 0.037542], [0,0,0,0], [9E9, 9E9, 9E9, 9E9, 9E9, 9E9]];
	VAR robtarget Openhole_1115 := [[442.05, -23.57, 180.74], [-0.008086, 0.707061, 0.705906, 0.04119], [0,0,0,0], [9E9, 9E9, 9E9, 9E9, 9E9, 9E9]];
	VAR robtarget Openhole_1116 := [[441.65, -23.86, 180.7], [-0.00847, 0.707056, 0.705765, 0.04354], [0,0,0,0], [9E9, 9E9, 9E9, 9E9, 9E9, 9E9]];
	VAR robtarget Openhole_1117 := [[441.23, -24.14, 180.66], [-0.008956, 0.70705, 0.705617, 0.045869], [0,0,0,0], [9E9, 9E9, 9E9, 9E9, 9E9, 9E9]];
	VAR robtarget Openhole_1118 := [[440.8, -24.39, 180.62], [-0.009568, 0.707042, 0.705464, 0.048165], [0,0,0,0], [9E9, 9E9, 9E9, 9E9, 9E9, 9E9]];
	VAR robtarget Openhole_1119 := [[439.91, -24.83, 180.53], [-0.011098, 0.70702, 0.705144, 0.052655], [0,0,0,0], [9E9, 9E9, 9E9, 9E9, 9E9, 9E9]];
	VAR robtarget Openhole_1120 := [[439.46, -25.04, 180.49], [-0.011919, 0.707006, 0.704974, 0.054876], [0,0,0,0], [9E9, 9E9, 9E9, 9E9, 9E9, 9E9]];
	VAR robtarget Openhole_1121 := [[438.55, -25.44, 180.39], [-0.013654, 0.706975, 0.704618, 0.059271], [0,0,0,0], [9E9, 9E9, 9E9, 9E9, 9E9, 9E9]];
	VAR robtarget Openhole_1122 := [[434.35, -26.98, 179.91], [-0.022668, 0.706743, 0.702756, 0.078317], [0,0,0,0], [9E9, 9E9, 9E9, 9E9, 9E9, 9E9]];
	VAR robtarget Openhole_1123 := [[432.92, -27.42, 179.74], [-0.026003, 0.706629, 0.70205, 0.084417], [0,0,0,0], [9E9, 9E9, 9E9, 9E9, 9E9, 9E9]];
	VAR robtarget Openhole_1124 := [[435.85, -24.75, 180.32], [-0.025085, 0.706662, 0.704029, 0.065902], [0,0,0,0], [9E9, 9E9, 9E9, 9E9, 9E9, 9E9]];
	VAR robtarget Openhole_1125 := [[437.63, -23.85, 180.52], [-0.022125, 0.706761, 0.704807, 0.056982], [0,0,0,0], [9E9, 9E9, 9E9, 9E9, 9E9, 9E9]];
	VAR robtarget Openhole_1126 := [[438.06, -23.61, 180.56], [-0.021452, 0.706781, 0.704986, 0.054721], [0,0,0,0], [9E9, 9E9, 9E9, 9E9, 9E9, 9E9]];
	VAR robtarget Openhole_1127 := [[439.34, -22.84, 180.69], [-0.019744, 0.706831, 0.705487, 0.047831], [0,0,0,0], [9E9, 9E9, 9E9, 9E9, 9E9, 9E9]];
	VAR robtarget Openhole_1128 := [[440.59, -22.01, 180.81], [-0.018332, 0.706869, 0.705926, 0.040843], [0,0,0,0], [9E9, 9E9, 9E9, 9E9, 9E9, 9E9]];
	VAR robtarget Openhole_1129 := [[441.01, -21.74, 180.84], [-0.017825, 0.706882, 0.706057, 0.038515], [0,0,0,0], [9E9, 9E9, 9E9, 9E9, 9E9, 9E9]];
	VAR robtarget Openhole_1130 := [[441.8, -21.35, 180.89], [-0.016474, 0.706915, 0.706264, 0.034522], [0,0,0,0], [9E9, 9E9, 9E9, 9E9, 9E9, 9E9]];
	VAR robtarget Openhole_1131 := [[438.17, -20.01, 180.96], [-0.033239, 0.706325, 0.705846, 0.042211], [0,0,0,0], [9E9, 9E9, 9E9, 9E9, 9E9, 9E9]];
	VAR robtarget Openhole_1132 := [[437.76, -20.3, 180.92], [-0.033645, 0.706306, 0.705702, 0.044549], [0,0,0,0], [9E9, 9E9, 9E9, 9E9, 9E9, 9E9]];
	VAR robtarget Openhole_1133 := [[436.96, -20.89, 180.84], [-0.034338, 0.706273, 0.705391, 0.049233], [0,0,0,0], [9E9, 9E9, 9E9, 9E9, 9E9, 9E9]];
	VAR robtarget Openhole_1134 := [[436.14, -21.45, 180.75], [-0.035199, 0.70623, 0.705052, 0.053873], [0,0,0,0], [9E9, 9E9, 9E9, 9E9, 9E9, 9E9]];
	VAR robtarget Openhole_1135 := [[435.72, -21.72, 180.71], [-0.035699, 0.706205, 0.704872, 0.056175], [0,0,0,0], [9E9, 9E9, 9E9, 9E9, 9E9, 9E9]];
	VAR robtarget Openhole_1136 := [[435.29, -21.98, 180.66], [-0.036241, 0.706177, 0.704686, 0.058461], [0,0,0,0], [9E9, 9E9, 9E9, 9E9, 9E9, 9E9]];
	VAR robtarget Openhole_1137 := [[434.43, -22.48, 180.57], [-0.037447, 0.706115, 0.704296, 0.06299], [0,0,0,0], [9E9, 9E9, 9E9, 9E9, 9E9, 9E9]];
	VAR robtarget Openhole_1138 := [[433.99, -22.72, 180.52], [-0.038116, 0.706079, 0.704092, 0.06523], [0,0,0,0], [9E9, 9E9, 9E9, 9E9, 9E9, 9E9]];
	VAR robtarget Openhole_1139 := [[433.55, -22.94, 180.47], [-0.038847, 0.706039, 0.703883, 0.067445], [0,0,0,0], [9E9, 9E9, 9E9, 9E9, 9E9, 9E9]];
	VAR robtarget Openhole_1140 := [[432.65, -23.37, 180.36], [-0.040434, 0.70595, 0.70345, 0.071819], [0,0,0,0], [9E9, 9E9, 9E9, 9E9, 9E9, 9E9]];
	VAR robtarget Openhole_1141 := [[432.19, -23.56, 180.31], [-0.041311, 0.705899, 0.703228, 0.073967], [0,0,0,0], [9E9, 9E9, 9E9, 9E9, 9E9, 9E9]];
	VAR robtarget Openhole_1142 := [[431.73, -23.75, 180.26], [-0.042227, 0.705845, 0.703001, 0.076093], [0,0,0,0], [9E9, 9E9, 9E9, 9E9, 9E9, 9E9]];
	VAR robtarget Openhole_1143 := [[430.8, -24.09, 180.16], [-0.044177, 0.705725, 0.702535, 0.080279], [0,0,0,0], [9E9, 9E9, 9E9, 9E9, 9E9, 9E9]];
	VAR robtarget Openhole_1144 := [[430.33, -24.25, 180.11], [-0.045224, 0.705659, 0.702298, 0.082329], [0,0,0,0], [9E9, 9E9, 9E9, 9E9, 9E9, 9E9]];
	VAR robtarget Openhole_1145 := [[427.45, -25.03, 179.8], [-0.052155, 0.705181, 0.700809, 0.094162], [0,0,0,0], [9E9, 9E9, 9E9, 9E9, 9E9, 9E9]];
	VAR robtarget Openhole_1146 := [[426.96, -25.13, 179.75], [-0.053405, 0.705087, 0.700552, 0.096057], [0,0,0,0], [9E9, 9E9, 9E9, 9E9, 9E9, 9E9]];
	VAR robtarget Openhole_1147 := [[425, -25.46, 179.55], [-0.058725, 0.704664, 0.699512, 0.103359], [0,0,0,0], [9E9, 9E9, 9E9, 9E9, 9E9, 9E9]];
	VAR robtarget Openhole_1148 := [[421.03, -25.86, 179.2], [-0.070271, 0.703606, 0.697369, 0.116944], [0,0,0,0], [9E9, 9E9, 9E9, 9E9, 9E9, 9E9]];
	VAR robtarget Openhole_1149 := [[416.05, -25.98, 178.83], [-0.085679, 0.701897, 0.694606, 0.132373], [0,0,0,0], [9E9, 9E9, 9E9, 9E9, 9E9, 9E9]];
	VAR robtarget Openhole_1150 := [[415.55, -25.97, 178.8], [-0.087251, 0.701703, 0.694325, 0.133837], [0,0,0,0], [9E9, 9E9, 9E9, 9E9, 9E9, 9E9]];
	VAR robtarget Openhole_1151 := [[401.58, -25.68, 178], [-0.129902, 0.695072, 0.685845, 0.172094], [0,0,0,0], [9E9, 9E9, 9E9, 9E9, 9E9, 9E9]];
	VAR robtarget Openhole_1152 := [[401.08, -25.68, 177.97], [-0.131317, 0.694806, 0.685513, 0.173412], [0,0,0,0], [9E9, 9E9, 9E9, 9E9, 9E9, 9E9]];
	VAR robtarget Openhole_1153 := [[395.6, -25.83, 177.54], [-0.146048, 0.69186, 0.681672, 0.187946], [0,0,0,0], [9E9, 9E9, 9E9, 9E9, 9E9, 9E9]];
	VAR robtarget Openhole_1154 := [[395.1, -25.86, 177.49], [-0.147304, 0.691593, 0.681304, 0.189273], [0,0,0,0], [9E9, 9E9, 9E9, 9E9, 9E9, 9E9]];
	VAR robtarget Openhole_1155 := [[394.33, -25.89, 177.43], [-0.149305, 0.691164, 0.680753, 0.191246], [0,0,0,0], [9E9, 9E9, 9E9, 9E9, 9E9, 9E9]];
	VAR robtarget Openhole_1156 := [[389.33, -25.89, 177.1], [-0.162456, 0.688192, 0.677244, 0.203322], [0,0,0,0], [9E9, 9E9, 9E9, 9E9, 9E9, 9E9]];
	VAR robtarget Openhole_1157 := [[362.33, -25.89, 177.18], [-0.183051, 0.683002, 0.683002, 0.183051], [0,0,0,0], [9E9, 9E9, 9E9, 9E9, 9E9, 9E9]];
	VAR robtarget Openhole_1158 := [[362.33, -25.1, 177.64], [-0.183051, 0.683002, 0.683002, 0.183051], [0,0,0,0], [9E9, 9E9, 9E9, 9E9, 9E9, 9E9]];
	VAR robtarget Openhole_1159 := [[389.33, -25.1, 177.55], [-0.164699, 0.687659, 0.677906, 0.201105], [0,0,0,0], [9E9, 9E9, 9E9, 9E9, 9E9, 9E9]];
	VAR robtarget Openhole_1160 := [[394.34, -25.1, 177.85], [-0.151604, 0.690664, 0.681388, 0.188973], [0,0,0,0], [9E9, 9E9, 9E9, 9E9, 9E9, 9E9]];
	VAR robtarget Openhole_1161 := [[395.22, -25.08, 177.91], [-0.149293, 0.691167, 0.682015, 0.186695], [0,0,0,0], [9E9, 9E9, 9E9, 9E9, 9E9, 9E9]];
	VAR robtarget Openhole_1162 := [[400.7, -24.87, 178.33], [-0.134821, 0.694135, 0.685869, 0.171999], [0,0,0,0], [9E9, 9E9, 9E9, 9E9, 9E9, 9E9]];
	VAR robtarget Openhole_1163 := [[402.2, -24.86, 178.41], [-0.130618, 0.694938, 0.686861, 0.167993], [0,0,0,0], [9E9, 9E9, 9E9, 9E9, 9E9, 9E9]];
	VAR robtarget Openhole_1164 := [[402.7, -24.86, 178.44], [-0.129191, 0.695205, 0.687186, 0.166661], [0,0,0,0], [9E9, 9E9, 9E9, 9E9, 9E9, 9E9]];
	VAR robtarget Openhole_1165 := [[416.18, -25.08, 179.13], [-0.088144, 0.701591, 0.695212, 0.129153], [0,0,0,0], [9E9, 9E9, 9E9, 9E9, 9E9, 9E9]];
	VAR robtarget Openhole_1166 := [[416.68, -25.08, 179.16], [-0.086588, 0.701785, 0.695488, 0.127659], [0,0,0,0], [9E9, 9E9, 9E9, 9E9, 9E9, 9E9]];
	VAR robtarget Openhole_1167 := [[422.16, -24.91, 179.52], [-0.069746, 0.703659, 0.698436, 0.110397], [0,0,0,0], [9E9, 9E9, 9E9, 9E9, 9E9, 9E9]];
	VAR robtarget Openhole_1168 := [[424.15, -24.72, 179.68], [-0.063942, 0.70421, 0.699476, 0.103603], [0,0,0,0], [9E9, 9E9, 9E9, 9E9, 9E9, 9E9]];
	VAR robtarget Openhole_1169 := [[425.13, -24.59, 179.76], [-0.061141, 0.704459, 0.699988, 0.100084], [0,0,0,0], [9E9, 9E9, 9E9, 9E9, 9E9, 9E9]];
	VAR robtarget Openhole_1170 := [[426.61, -24.36, 179.89], [-0.057088, 0.704799, 0.700744, 0.094644], [0,0,0,0], [9E9, 9E9, 9E9, 9E9, 9E9, 9E9]];
	VAR robtarget Openhole_1171 := [[427.1, -24.27, 179.94], [-0.055798, 0.704902, 0.700994, 0.092776], [0,0,0,0], [9E9, 9E9, 9E9, 9E9, 9E9, 9E9]];
	VAR robtarget Openhole_1172 := [[428.07, -24.05, 180.03], [-0.053315, 0.705094, 0.701489, 0.088957], [0,0,0,0], [9E9, 9E9, 9E9, 9E9, 9E9, 9E9]];
	VAR robtarget Openhole_1173 := [[429.52, -23.69, 180.17], [-0.04975, 0.705354, 0.702208, 0.083087], [0,0,0,0], [9E9, 9E9, 9E9, 9E9, 9E9, 9E9]];
	VAR robtarget Openhole_1174 := [[430.48, -23.42, 180.26], [-0.047494, 0.70551, 0.702671, 0.079076], [0,0,0,0], [9E9, 9E9, 9E9, 9E9, 9E9, 9E9]];
	VAR robtarget Openhole_1175 := [[428.63, -22.36, 180.4], [-0.057111, 0.704797, 0.702389, 0.081549], [0,0,0,0], [9E9, 9E9, 9E9, 9E9, 9E9, 9E9]];
	VAR robtarget Openhole_1176 := [[428.14, -22.45, 180.36], [-0.0584, 0.704691, 0.702166, 0.083445], [0,0,0,0], [9E9, 9E9, 9E9, 9E9, 9E9, 9E9]];
	VAR robtarget Openhole_1177 := [[425.18, -22.88, 180.16], [-0.066638, 0.70396, 0.700786, 0.094332], [0,0,0,0], [9E9, 9E9, 9E9, 9E9, 9E9, 9E9]];
	VAR robtarget Openhole_1178 := [[420.69, -23.18, 179.92], [-0.080065, 0.702559, 0.698604, 0.109327], [0,0,0,0], [9E9, 9E9, 9E9, 9E9, 9E9, 9E9]];
	VAR robtarget Openhole_1179 := [[418.2, -23.21, 179.81], [-0.087848, 0.701629, 0.697346, 0.117084], [0,0,0,0], [9E9, 9E9, 9E9, 9E9, 9E9, 9E9]];
	VAR robtarget Openhole_1180 := [[417.7, -23.21, 179.79], [-0.089414, 0.701431, 0.69709, 0.1186], [0,0,0,0], [9E9, 9E9, 9E9, 9E9, 9E9, 9E9]];
	VAR robtarget Openhole_1181 := [[417.2, -23.21, 179.77], [-0.090972, 0.70123, 0.69683, 0.120115], [0,0,0,0], [9E9, 9E9, 9E9, 9E9, 9E9, 9E9]];
	VAR robtarget Openhole_1182 := [[416.7, -23.21, 179.75], [-0.09254, 0.701025, 0.696571, 0.12161], [0,0,0,0], [9E9, 9E9, 9E9, 9E9, 9E9, 9E9]];
	VAR robtarget Openhole_1183 := [[404.71, -23.06, 179.33], [-0.128943, 0.695251, 0.689744, 0.155736], [0,0,0,0], [9E9, 9E9, 9E9, 9E9, 9E9, 9E9]];
	VAR robtarget Openhole_1184 := [[404.21, -23.06, 179.31], [-0.130375, 0.694984, 0.689432, 0.157111], [0,0,0,0], [9E9, 9E9, 9E9, 9E9, 9E9, 9E9]];
	VAR robtarget Openhole_1185 := [[397.22, -23.22, 178.96], [-0.149375, 0.691149, 0.684804, 0.176192], [0,0,0,0], [9E9, 9E9, 9E9, 9E9, 9E9, 9E9]];
	VAR robtarget Openhole_1186 := [[395.23, -23.34, 178.82], [-0.154394, 0.690045, 0.683385, 0.181619], [0,0,0,0], [9E9, 9E9, 9E9, 9E9, 9E9, 9E9]];
	VAR robtarget Openhole_1187 := [[394.34, -23.36, 178.77], [-0.156684, 0.689529, 0.682765, 0.183936], [0,0,0,0], [9E9, 9E9, 9E9, 9E9, 9E9, 9E9]];
	VAR robtarget Openhole_1188 := [[389.34, -23.36, 178.56], [-0.169655, 0.686453, 0.679344, 0.196195], [0,0,0,0], [9E9, 9E9, 9E9, 9E9, 9E9, 9E9]];
	VAR robtarget Openhole_1189 := [[362.34, -23.36, 178.64], [-0.183051, 0.683002, 0.683002, 0.183051], [0,0,0,0], [9E9, 9E9, 9E9, 9E9, 9E9, 9E9]];
	VAR robtarget Openhole_1190 := [[362.34, -22.46, 179.16], [-0.183051, 0.683002, 0.683002, 0.183051], [0,0,0,0], [9E9, 9E9, 9E9, 9E9, 9E9, 9E9]];
	VAR robtarget Openhole_1191 := [[389.34, -22.46, 179.08], [-0.172229, 0.685811, 0.680077, 0.193637], [0,0,0,0], [9E9, 9E9, 9E9, 9E9, 9E9, 9E9]];
	VAR robtarget Openhole_1192 := [[394.34, -22.46, 179.24], [-0.159322, 0.688924, 0.683466, 0.181313], [0,0,0,0], [9E9, 9E9, 9E9, 9E9, 9E9, 9E9]];
	VAR robtarget Openhole_1193 := [[395.12, -22.43, 179.28], [-0.157343, 0.689379, 0.68401, 0.179251], [0,0,0,0], [9E9, 9E9, 9E9, 9E9, 9E9, 9E9]];
	VAR robtarget Openhole_1194 := [[401.6, -22.16, 179.62], [-0.140478, 0.693012, 0.688424, 0.161468], [0,0,0,0], [9E9, 9E9, 9E9, 9E9, 9E9, 9E9]];
	VAR robtarget Openhole_1195 := [[405.6, -22.12, 179.76], [-0.129249, 0.695194, 0.690928, 0.150393], [0,0,0,0], [9E9, 9E9, 9E9, 9E9, 9E9, 9E9]];
	VAR robtarget Openhole_1196 := [[406.1, -22.12, 179.77], [-0.127806, 0.695461, 0.69123, 0.148999], [0,0,0,0], [9E9, 9E9, 9E9, 9E9, 9E9, 9E9]];
	VAR robtarget Openhole_1197 := [[418.1, -22.26, 180.09], [-0.091215, 0.701199, 0.697799, 0.11435], [0,0,0,0], [9E9, 9E9, 9E9, 9E9, 9E9, 9E9]];
	VAR robtarget Openhole_1198 := [[418.6, -22.26, 180.1], [-0.089652, 0.7014, 0.698048, 0.112823], [0,0,0,0], [9E9, 9E9, 9E9, 9E9, 9E9, 9E9]];
	VAR robtarget Openhole_1199 := [[423.09, -22.18, 180.26], [-0.075664, 0.703047, 0.700197, 0.098613], [0,0,0,0], [9E9, 9E9, 9E9, 9E9, 9E9, 9E9]];
	VAR robtarget Openhole_1200 := [[427.57, -21.76, 180.49], [-0.062567, 0.704333, 0.702218, 0.083001], [0,0,0,0], [9E9, 9E9, 9E9, 9E9, 9E9, 9E9]];
	VAR robtarget Openhole_1201 := [[428.06, -21.68, 180.52], [-0.061206, 0.704453, 0.702434, 0.08116], [0,0,0,0], [9E9, 9E9, 9E9, 9E9, 9E9, 9E9]];
	VAR robtarget Openhole_1202 := [[429.04, -21.5, 180.58], [-0.058585, 0.704676, 0.702859, 0.077388], [0,0,0,0], [9E9, 9E9, 9E9, 9E9, 9E9, 9E9]];
	VAR robtarget Openhole_1203 := [[430.01, -21.29, 180.64], [-0.056106, 0.704877, 0.703277, 0.073499], [0,0,0,0], [9E9, 9E9, 9E9, 9E9, 9E9, 9E9]];
	VAR robtarget Openhole_1204 := [[432.42, -20.64, 180.8], [-0.0503, 0.705315, 0.704254, 0.063448], [0,0,0,0], [9E9, 9E9, 9E9, 9E9, 9E9, 9E9]];
	VAR robtarget Openhole_1205 := [[433.85, -20.18, 180.89], [-0.047116, 0.705535, 0.70479, 0.057194], [0,0,0,0], [9E9, 9E9, 9E9, 9E9, 9E9, 9E9]];
	VAR robtarget Openhole_1206 := [[434.32, -20.01, 180.92], [-0.046141, 0.7056, 0.70496, 0.055059], [0,0,0,0], [9E9, 9E9, 9E9, 9E9, 9E9, 9E9]];
	VAR robtarget Openhole_1207 := [[434.78, -19.82, 180.95], [-0.045238, 0.705658, 0.705126, 0.052888], [0,0,0,0], [9E9, 9E9, 9E9, 9E9, 9E9, 9E9]];
	VAR robtarget Openhole_1208 := [[435.69, -19.42, 181.01], [-0.043543, 0.705765, 0.705442, 0.048489], [0,0,0,0], [9E9, 9E9, 9E9, 9E9, 9E9, 9E9]];
	VAR robtarget Openhole_1209 := [[436.63, -19.07, 181.06], [-0.041575, 0.705883, 0.705725, 0.044189], [0,0,0,0], [9E9, 9E9, 9E9, 9E9, 9E9, 9E9]];
	VAR robtarget Openhole_1210 := [[437.08, -18.86, 181.08], [-0.040786, 0.70593, 0.705861, 0.041954], [0,0,0,0], [9E9, 9E9, 9E9, 9E9, 9E9, 9E9]];
	VAR robtarget Openhole_1211 := [[436.53, -17.57, 181.24], [-0.046931, 0.705548, 0.706005, 0.039449], [0,0,0,0], [9E9, 9E9, 9E9, 9E9, 9E9, 9E9]];
	VAR robtarget Openhole_1212 := [[435.53, -17.56, 181.26], [-0.050291, 0.705316, 0.705812, 0.042771], [0,0,0,0], [9E9, 9E9, 9E9, 9E9, 9E9, 9E9]];
	VAR robtarget Openhole_1213 := [[435.04, -17.58, 181.26], [-0.05189, 0.7052, 0.705705, 0.044505], [0,0,0,0], [9E9, 9E9, 9E9, 9E9, 9E9, 9E9]];
	VAR robtarget Openhole_1214 := [[434.54, -17.58, 181.27], [-0.053553, 0.705076, 0.705598, 0.046172], [0,0,0,0], [9E9, 9E9, 9E9, 9E9, 9E9, 9E9]];
	VAR robtarget Openhole_1215 := [[434.04, -17.59, 181.27], [-0.055198, 0.704949, 0.705486, 0.047851], [0,0,0,0], [9E9, 9E9, 9E9, 9E9, 9E9, 9E9]];
	VAR robtarget Openhole_1216 := [[433.54, -17.58, 181.28], [-0.05688, 0.704815, 0.705373, 0.049488], [0,0,0,0], [9E9, 9E9, 9E9, 9E9, 9E9, 9E9]];
	VAR robtarget Openhole_1217 := [[433.04, -17.58, 181.29], [-0.058511, 0.704682, 0.705253, 0.051171], [0,0,0,0], [9E9, 9E9, 9E9, 9E9, 9E9, 9E9]];
	VAR robtarget Openhole_1218 := [[432.54, -17.58, 181.29], [-0.060164, 0.704543, 0.705131, 0.052826], [0,0,0,0], [9E9, 9E9, 9E9, 9E9, 9E9, 9E9]];
	VAR robtarget Openhole_1219 := [[418.04, -17.3, 181.58], [-0.107378, 0.698906, 0.700209, 0.098527], [0,0,0,0], [9E9, 9E9, 9E9, 9E9, 9E9, 9E9]];
	VAR robtarget Openhole_1220 := [[408.54, -17.2, 181.78], [-0.136002, 0.693904, 0.695647, 0.126787], [0,0,0,0], [9E9, 9E9, 9E9, 9E9, 9E9, 9E9]];
	VAR robtarget Openhole_1221 := [[408.04, -17.2, 181.79], [-0.137436, 0.693622, 0.69538, 0.128245], [0,0,0,0], [9E9, 9E9, 9E9, 9E9, 9E9, 9E9]];
	VAR robtarget Openhole_1222 := [[398.55, -17.4, 181.86], [-0.163121, 0.688034, 0.689814, 0.155424], [0,0,0,0], [9E9, 9E9, 9E9, 9E9, 9E9, 9E9]];
	VAR robtarget Openhole_1223 := [[394.35, -17.6, 181.82], [-0.173517, 0.685487, 0.687076, 0.167113], [0,0,0,0], [9E9, 9E9, 9E9, 9E9, 9E9, 9E9]];
	VAR robtarget Openhole_1224 := [[362.35, -17.6, 181.97], [-0.183051, 0.683002, 0.683002, 0.183051], [0,0,0,0], [9E9, 9E9, 9E9, 9E9, 9E9, 9E9]];
	VAR robtarget Openhole_1225 := [[362.35, -18.56, 181.42], [-0.183051, 0.683002, 0.683002, 0.183051], [0,0,0,0], [9E9, 9E9, 9E9, 9E9, 9E9, 9E9]];
	VAR robtarget Openhole_1226 := [[389.35, -18.56, 181.33], [-0.183342, 0.682924, 0.683141, 0.182533], [0,0,0,0], [9E9, 9E9, 9E9, 9E9, 9E9, 9E9]];
	VAR robtarget Openhole_1227 := [[394.35, -18.56, 181.31], [-0.170717, 0.686189, 0.686386, 0.169925], [0,0,0,0], [9E9, 9E9, 9E9, 9E9, 9E9, 9E9]];
	VAR robtarget Openhole_1228 := [[402.43, -18.22, 181.42], [-0.150108, 0.69099, 0.691591, 0.147317], [0,0,0,0], [9E9, 9E9, 9E9, 9E9, 9E9, 9E9]];
	VAR robtarget Openhole_1229 := [[408.43, -18.16, 181.4], [-0.133355, 0.694418, 0.695034, 0.130108], [0,0,0,0], [9E9, 9E9, 9E9, 9E9, 9E9, 9E9]];
	VAR robtarget Openhole_1230 := [[408.93, -18.16, 181.4], [-0.131903, 0.694695, 0.695303, 0.12866], [0,0,0,0], [9E9, 9E9, 9E9, 9E9, 9E9, 9E9]];
	VAR robtarget Openhole_1231 := [[426.43, -18.45, 181.19], [-0.077227, 0.702877, 0.703042, 0.07571], [0,0,0,0], [9E9, 9E9, 9E9, 9E9, 9E9, 9E9]];
	VAR robtarget Openhole_1232 := [[426.93, -18.44, 181.19], [-0.07562, 0.703052, 0.703215, 0.074087], [0,0,0,0], [9E9, 9E9, 9E9, 9E9, 9E9, 9E9]];
	VAR robtarget Openhole_1233 := [[430.42, -18.38, 181.18], [-0.064432, 0.704165, 0.704342, 0.062474], [0,0,0,0], [9E9, 9E9, 9E9, 9E9, 9E9, 9E9]];
	VAR robtarget Openhole_1234 := [[431.42, -18.38, 181.17], [-0.061145, 0.704458, 0.704625, 0.059186], [0,0,0,0], [9E9, 9E9, 9E9, 9E9, 9E9, 9E9]];
	VAR robtarget Openhole_1235 := [[431.92, -18.36, 181.17], [-0.0596, 0.704591, 0.70477, 0.057441], [0,0,0,0], [9E9, 9E9, 9E9, 9E9, 9E9, 9E9]];
	VAR robtarget Openhole_1236 := [[433.09, -19.64, 180.97], [-0.051447, 0.705233, 0.704733, 0.05789], [0,0,0,0], [9E9, 9E9, 9E9, 9E9, 9E9, 9E9]];
	VAR robtarget Openhole_1237 := [[431.14, -20.07, 180.88], [-0.056453, 0.70485, 0.704042, 0.065766], [0,0,0,0], [9E9, 9E9, 9E9, 9E9, 9E9, 9E9]];
	VAR robtarget Openhole_1238 := [[429.67, -20.35, 180.81], [-0.06036, 0.704526, 0.703481, 0.071516], [0,0,0,0], [9E9, 9E9, 9E9, 9E9, 9E9, 9E9]];
	VAR robtarget Openhole_1239 := [[429.17, -20.43, 180.79], [-0.061722, 0.704408, 0.703289, 0.07338], [0,0,0,0], [9E9, 9E9, 9E9, 9E9, 9E9, 9E9]];
	VAR robtarget Openhole_1240 := [[428.18, -20.56, 180.75], [-0.064537, 0.704156, 0.702899, 0.077022], [0,0,0,0], [9E9, 9E9, 9E9, 9E9, 9E9, 9E9]];
	VAR robtarget Openhole_1241 := [[426.19, -20.74, 180.68], [-0.070413, 0.703592, 0.702096, 0.084034], [0,0,0,0], [9E9, 9E9, 9E9, 9E9, 9E9, 9E9]];
	VAR robtarget Openhole_1242 := [[425.2, -20.8, 180.65], [-0.073423, 0.703285, 0.70168, 0.087438], [0,0,0,0], [9E9, 9E9, 9E9, 9E9, 9E9, 9E9]];
	VAR robtarget Openhole_1243 := [[421.2, -20.9, 180.55], [-0.085891, 0.701871, 0.699948, 0.10036], [0,0,0,0], [9E9, 9E9, 9E9, 9E9, 9E9, 9E9]];
	VAR robtarget Openhole_1244 := [[420.7, -20.89, 180.55], [-0.087477, 0.701675, 0.699724, 0.101912], [0,0,0,0], [9E9, 9E9, 9E9, 9E9, 9E9, 9E9]];
	VAR robtarget Openhole_1245 := [[406.7, -20.73, 180.36], [-0.130385, 0.694982, 0.692491, 0.143024], [0,0,0,0], [9E9, 9E9, 9E9, 9E9, 9E9, 9E9]];
	VAR robtarget Openhole_1246 := [[406.2, -20.73, 180.36], [-0.131822, 0.694711, 0.692198, 0.144438], [0,0,0,0], [9E9, 9E9, 9E9, 9E9, 9E9, 9E9]];
	VAR robtarget Openhole_1247 := [[398.21, -20.89, 180.14], [-0.153634, 0.690215, 0.687168, 0.166734], [0,0,0,0], [9E9, 9E9, 9E9, 9E9, 9E9, 9E9]];
	VAR robtarget Openhole_1248 := [[395.21, -21.06, 180], [-0.16113, 0.688504, 0.685109, 0.175002], [0,0,0,0], [9E9, 9E9, 9E9, 9E9, 9E9, 9E9]];
	VAR robtarget Openhole_1249 := [[394.34, -21.09, 179.97], [-0.163327, 0.687986, 0.684512, 0.177321], [0,0,0,0], [9E9, 9E9, 9E9, 9E9, 9E9, 9E9]];
	VAR robtarget Openhole_1250 := [[389.34, -21.09, 179.87], [-0.176135, 0.684819, 0.681173, 0.189745], [0,0,0,0], [9E9, 9E9, 9E9, 9E9, 9E9, 9E9]];
	VAR robtarget Openhole_1251 := [[362.34, -21.09, 179.95], [-0.183051, 0.683002, 0.683002, 0.183051], [0,0,0,0], [9E9, 9E9, 9E9, 9E9, 9E9, 9E9]];
	VAR robtarget Openhole_1252 := [[362.35, -15.88, 182.97], [-0.183051, 0.683002, 0.683002, 0.183051], [0,0,0,0], [9E9, 9E9, 9E9, 9E9, 9E9, 9E9]];
	VAR robtarget Openhole_1253 := [[389.35, -15.88, 182.88], [-0.190955, 0.680835, 0.685142, 0.174871], [0,0,0,0], [9E9, 9E9, 9E9, 9E9, 9E9, 9E9]];
	VAR robtarget Openhole_1254 := [[394.35, -15.88, 182.73], [-0.178524, 0.6842, 0.688283, 0.162069], [0,0,0,0], [9E9, 9E9, 9E9, 9E9, 9E9, 9E9]];
	VAR robtarget Openhole_1255 := [[402.84, -15.53, 182.63], [-0.15713, 0.689427, 0.693514, 0.137979], [0,0,0,0], [9E9, 9E9, 9E9, 9E9, 9E9, 9E9]];
	VAR robtarget Openhole_1256 := [[411.34, -15.42, 182.38], [-0.133449, 0.6944, 0.698026, 0.112959], [0,0,0,0], [9E9, 9E9, 9E9, 9E9, 9E9, 9E9]];
	VAR robtarget Openhole_1257 := [[411.84, -15.42, 182.36], [-0.131987, 0.694679, 0.698267, 0.111462], [0,0,0,0], [9E9, 9E9, 9E9, 9E9, 9E9, 9E9]];
	VAR robtarget Openhole_1258 := [[425.83, -15.62, 181.83], [-0.088457, 0.701552, 0.7038, 0.06831], [0,0,0,0], [9E9, 9E9, 9E9, 9E9, 9E9, 9E9]];
	VAR robtarget Openhole_1259 := [[433.81, -16, 181.51], [-0.061259, 0.704448, 0.705782, 0.04327], [0,0,0,0], [9E9, 9E9, 9E9, 9E9, 9E9, 9E9]];
	VAR robtarget Openhole_1260 := [[434.8, -16.09, 181.47], [-0.057652, 0.704753, 0.70596, 0.040264], [0,0,0,0], [9E9, 9E9, 9E9, 9E9, 9E9, 9E9]];
	VAR robtarget Openhole_1261 := [[435.3, -16.15, 181.45], [-0.05581, 0.704901, 0.706041, 0.038801], [0,0,0,0], [9E9, 9E9, 9E9, 9E9, 9E9, 9E9]];
	VAR robtarget Openhole_1262 := [[438.22, -12.1, 181.8], [-0.059738, 0.704579, 0.706942, 0.015284], [0,0,0,0], [9E9, 9E9, 9E9, 9E9, 9E9, 9E9]];
	VAR robtarget Openhole_1263 := [[439.21, -12.15, 181.73], [-0.056234, 0.704867, 0.707003, 0.012091], [0,0,0,0], [9E9, 9E9, 9E9, 9E9, 9E9, 9E9]];
	VAR robtarget Openhole_1264 := [[440.21, -12.22, 181.66], [-0.052664, 0.705143, 0.70705, 0.008959], [0,0,0,0], [9E9, 9E9, 9E9, 9E9, 9E9, 9E9]];
	VAR robtarget Openhole_1265 := [[441.7, -12.31, 181.56], [-0.047366, 0.705519, 0.707095, 0.004167], [0,0,0,0], [9E9, 9E9, 9E9, 9E9, 9E9, 9E9]];
	VAR robtarget Openhole_1266 := [[442.2, -12.35, 181.52], [-0.045565, 0.705637, 0.707102, 0.002604], [0,0,0,0], [9E9, 9E9, 9E9, 9E9, 9E9, 9E9]];
	VAR robtarget Openhole_1267 := [[443.19, -12.46, 181.45], [-0.041857, 0.705867, 0.707107, -0.000401], [0,0,0,0], [9E9, 9E9, 9E9, 9E9, 9E9, 9E9]];
	VAR robtarget Openhole_1268 := [[443.92, -12.82, 181.39], [-0.038169, 0.706076, 0.707105, -0.001667], [0,0,0,0], [9E9, 9E9, 9E9, 9E9, 9E9, 9E9]];
	VAR robtarget Openhole_1269 := [[455.86, -14.06, 180.75], [0.006547, 0.707076, 0.706079, -0.038102], [0,0,0,0], [9E9, 9E9, 9E9, 9E9, 9E9, 9E9]];
	VAR robtarget Openhole_1270 := [[456.33, -13.69, 180.7], [0.006879, 0.707073, 0.70592, -0.040942], [0,0,0,0], [9E9, 9E9, 9E9, 9E9, 9E9, 9E9]];
	VAR robtarget Openhole_1271 := [[456.73, -13.4, 180.66], [0.007261, 0.70707, 0.70578, -0.043295], [0,0,0,0], [9E9, 9E9, 9E9, 9E9, 9E9, 9E9]];
	VAR robtarget Openhole_1272 := [[457.15, -13.13, 180.62], [0.007774, 0.707064, 0.705634, -0.04562], [0,0,0,0], [9E9, 9E9, 9E9, 9E9, 9E9, 9E9]];
	VAR robtarget Openhole_1273 := [[457.59, -12.89, 180.57], [0.008461, 0.707056, 0.705483, -0.047896], [0,0,0,0], [9E9, 9E9, 9E9, 9E9, 9E9, 9E9]];
	VAR robtarget Openhole_1274 := [[458.49, -12.46, 180.48], [0.010048, 0.707035, 0.705165, -0.052371], [0,0,0,0], [9E9, 9E9, 9E9, 9E9, 9E9, 9E9]];
	VAR robtarget Openhole_1275 := [[459.4, -12.06, 180.39], [0.011795, 0.707008, 0.704824, -0.056772], [0,0,0,0], [9E9, 9E9, 9E9, 9E9, 9E9, 9E9]];
	VAR robtarget Openhole_1276 := [[461.72, -11.18, 180.13], [0.016668, 0.70691, 0.703878, -0.067497], [0,0,0,0], [9E9, 9E9, 9E9, 9E9, 9E9, 9E9]];
	VAR robtarget Openhole_1277 := [[464.08, -10.39, 179.84], [0.021976, 0.706765, 0.702802, -0.077905], [0,0,0,0], [9E9, 9E9, 9E9, 9E9, 9E9, 9E9]];
	VAR robtarget Openhole_1278 := [[465.51, -9.96, 179.65], [0.025332, 0.706653, 0.702099, -0.084002], [0,0,0,0], [9E9, 9E9, 9E9, 9E9, 9E9, 9E9]];
	VAR robtarget Openhole_1279 := [[468.4, -7.76, 178.99], [0.027737, 0.706563, 0.699909, -0.100636], [0,0,0,0], [9E9, 9E9, 9E9, 9E9, 9E9, 9E9]];
	VAR robtarget Openhole_1280 := [[460.65, -9.48, 180.02], [0.007351, 0.707069, 0.703669, -0.06964], [0,0,0,0], [9E9, 9E9, 9E9, 9E9, 9E9, 9E9]];
	VAR robtarget Openhole_1281 := [[457.75, -10.16, 180.34], [-0.000183, 0.707107, 0.704754, -0.057639], [0,0,0,0], [9E9, 9E9, 9E9, 9E9, 9E9, 9E9]];
	VAR robtarget Openhole_1282 := [[456.79, -10.4, 180.44], [-0.00268, 0.707102, 0.705072, -0.0536], [0,0,0,0], [9E9, 9E9, 9E9, 9E9, 9E9, 9E9]];
	VAR robtarget Openhole_1283 := [[456.31, -10.53, 180.49], [-0.003883, 0.707096, 0.705225, -0.05155], [0,0,0,0], [9E9, 9E9, 9E9, 9E9, 9E9, 9E9]];
	VAR robtarget Openhole_1284 := [[455.82, -10.65, 180.54], [-0.005124, 0.707088, 0.705371, -0.049518], [0,0,0,0], [9E9, 9E9, 9E9, 9E9, 9E9, 9E9]];
	VAR robtarget Openhole_1285 := [[454.86, -10.92, 180.63], [-0.007471, 0.707067, 0.70565, -0.045369], [0,0,0,0], [9E9, 9E9, 9E9, 9E9, 9E9, 9E9]];
	VAR robtarget Openhole_1286 := [[454.39, -11.08, 180.68], [-0.008533, 0.707055, 0.705784, -0.043233], [0,0,0,0], [9E9, 9E9, 9E9, 9E9, 9E9, 9E9]];
	VAR robtarget Openhole_1287 := [[453.93, -11.26, 180.72], [-0.009469, 0.707043, 0.705915, -0.041036], [0,0,0,0], [9E9, 9E9, 9E9, 9E9, 9E9, 9E9]];
	VAR robtarget Openhole_1288 := [[453.3, -11.75, 180.78], [-0.009967, 0.707037, 0.706124, -0.037275], [0,0,0,0], [9E9, 9E9, 9E9, 9E9, 9E9, 9E9]];
	VAR robtarget Openhole_1289 := [[446.72, -11.14, 181.26], [-0.034375, 0.706271, 0.706905, -0.016899], [0,0,0,0], [9E9, 9E9, 9E9, 9E9, 9E9, 9E9]];
	VAR robtarget Openhole_1290 := [[446.16, -10.86, 181.31], [-0.037242, 0.706125, 0.706926, -0.015968], [0,0,0,0], [9E9, 9E9, 9E9, 9E9, 9E9, 9E9]];
	VAR robtarget Openhole_1291 := [[445.18, -10.67, 181.4], [-0.041171, 0.705907, 0.706983, -0.013245], [0,0,0,0], [9E9, 9E9, 9E9, 9E9, 9E9, 9E9]];
	VAR robtarget Openhole_1292 := [[444.69, -10.59, 181.44], [-0.043103, 0.705792, 0.707008, -0.011842], [0,0,0,0], [9E9, 9E9, 9E9, 9E9, 9E9, 9E9]];
	VAR robtarget Openhole_1293 := [[444.19, -10.54, 181.48], [-0.044948, 0.705677, 0.707031, -0.010326], [0,0,0,0], [9E9, 9E9, 9E9, 9E9, 9E9, 9E9]];
	VAR robtarget Openhole_1294 := [[443.69, -10.51, 181.52], [-0.046722, 0.705562, 0.707053, -0.008727], [0,0,0,0], [9E9, 9E9, 9E9, 9E9, 9E9, 9E9]];
	VAR robtarget Openhole_1295 := [[442.7, -10.49, 181.61], [-0.050141, 0.705327, 0.707086, -0.005394], [0,0,0,0], [9E9, 9E9, 9E9, 9E9, 9E9, 9E9]];
	VAR robtarget Openhole_1296 := [[439.21, -10.53, 181.89], [-0.061671, 0.704412, 0.707076, 0.006632], [0,0,0,0], [9E9, 9E9, 9E9, 9E9, 9E9, 9E9]];
	VAR robtarget Openhole_1297 := [[438.71, -10.53, 181.93], [-0.063331, 0.704265, 0.707058, 0.008325], [0,0,0,0], [9E9, 9E9, 9E9, 9E9, 9E9, 9E9]];
	VAR robtarget Openhole_1298 := [[438.21, -10.53, 181.97], [-0.064992, 0.704114, 0.707036, 0.010012], [0,0,0,0], [9E9, 9E9, 9E9, 9E9, 9E9, 9E9]];
	VAR robtarget Openhole_1299 := [[437.71, -10.53, 182.01], [-0.066645, 0.703959, 0.70701, 0.011705], [0,0,0,0], [9E9, 9E9, 9E9, 9E9, 9E9, 9E9]];
	VAR robtarget Openhole_1300 := [[437.22, -10.53, 182.05], [-0.068312, 0.703799, 0.70698, 0.013379], [0,0,0,0], [9E9, 9E9, 9E9, 9E9, 9E9, 9E9]];
	VAR robtarget Openhole_1301 := [[438.63, -8.96, 182.1], [-0.068879, 0.703744, 0.707099, 0.003312], [0,0,0,0], [9E9, 9E9, 9E9, 9E9, 9E9, 9E9]];
	VAR robtarget Openhole_1302 := [[444.58, -8.42, 181.55], [-0.050762, 0.705282, 0.706857, -0.018788], [0,0,0,0], [9E9, 9E9, 9E9, 9E9, 9E9, 9E9]];
	VAR robtarget Openhole_1303 := [[445.07, -8.4, 181.5], [-0.049175, 0.705395, 0.706807, -0.020574], [0,0,0,0], [9E9, 9E9, 9E9, 9E9, 9E9, 9E9]];
	VAR robtarget Openhole_1304 := [[446.56, -8.37, 181.35], [-0.044243, 0.705721, 0.706637, -0.025773], [0,0,0,0], [9E9, 9E9, 9E9, 9E9, 9E9, 9E9]];
	VAR robtarget Openhole_1305 := [[447.06, -8.37, 181.3], [-0.04255, 0.705825, 0.706573, -0.02746], [0,0,0,0], [9E9, 9E9, 9E9, 9E9, 9E9, 9E9]];
	VAR robtarget Openhole_1306 := [[452.53, -8.5, 180.74], [-0.023533, 0.706715, 0.705633, -0.045625], [0,0,0,0], [9E9, 9E9, 9E9, 9E9, 9E9, 9E9]];
	VAR robtarget Openhole_1307 := [[453.03, -8.5, 180.69], [-0.021846, 0.706769, 0.705522, -0.047317], [0,0,0,0], [9E9, 9E9, 9E9, 9E9, 9E9, 9E9]];
	VAR robtarget Openhole_1308 := [[453.53, -8.5, 180.64], [-0.020169, 0.706819, 0.705406, -0.049016], [0,0,0,0], [9E9, 9E9, 9E9, 9E9, 9E9, 9E9]];
	VAR robtarget Openhole_1309 := [[454.02, -8.5, 180.59], [-0.01847, 0.706866, 0.705287, -0.050694], [0,0,0,0], [9E9, 9E9, 9E9, 9E9, 9E9, 9E9]];
	VAR robtarget Openhole_1310 := [[454.52, -8.49, 180.54], [-0.016799, 0.706907, 0.705163, -0.052395], [0,0,0,0], [9E9, 9E9, 9E9, 9E9, 9E9, 9E9]];
	VAR robtarget Openhole_1311 := [[455.02, -8.48, 180.49], [-0.015149, 0.706944, 0.705033, -0.054115], [0,0,0,0], [9E9, 9E9, 9E9, 9E9, 9E9, 9E9]];
	VAR robtarget Openhole_1312 := [[457, -8.37, 180.28], [-0.008764, 0.707052, 0.704456, -0.061169], [0,0,0,0], [9E9, 9E9, 9E9, 9E9, 9E9, 9E9]];
	VAR robtarget Openhole_1313 := [[454.64, -6.86, 180.44], [-0.02187, 0.706768, 0.704704, -0.058239], [0,0,0,0], [9E9, 9E9, 9E9, 9E9, 9E9, 9E9]];
	VAR robtarget Openhole_1314 := [[453.64, -6.78, 180.55], [-0.025505, 0.706647, 0.704952, -0.055159], [0,0,0,0], [9E9, 9E9, 9E9, 9E9, 9E9, 9E9]];
	VAR robtarget Openhole_1315 := [[452.66, -6.67, 180.67], [-0.029251, 0.706501, 0.705177, -0.052208], [0,0,0,0], [9E9, 9E9, 9E9, 9E9, 9E9, 9E9]];
	VAR robtarget Openhole_1316 := [[449.69, -6.4, 181.02], [-0.040232, 0.705961, 0.705796, -0.043034], [0,0,0,0], [9E9, 9E9, 9E9, 9E9, 9E9, 9E9]];
	VAR robtarget Openhole_1317 := [[448.2, -6.35, 181.2], [-0.045463, 0.705644, 0.706077, -0.038152], [0,0,0,0], [9E9, 9E9, 9E9, 9E9, 9E9, 9E9]];
	VAR robtarget Openhole_1318 := [[447.71, -6.35, 181.26], [-0.047121, 0.705535, 0.706167, -0.036438], [0,0,0,0], [9E9, 9E9, 9E9, 9E9, 9E9, 9E9]];
	VAR robtarget Openhole_1319 := [[447.21, -6.37, 181.32], [-0.048749, 0.705424, 0.706255, -0.034694], [0,0,0,0], [9E9, 9E9, 9E9, 9E9, 9E9, 9E9]];
	VAR robtarget Openhole_1320 := [[446.22, -6.44, 181.44], [-0.051859, 0.705203, 0.706424, -0.031076], [0,0,0,0], [9E9, 9E9, 9E9, 9E9, 9E9, 9E9]];
	VAR robtarget Openhole_1321 := [[445.23, -6.56, 181.55], [-0.054764, 0.704983, 0.70658, -0.02729], [0,0,0,0], [9E9, 9E9, 9E9, 9E9, 9E9, 9E9]];
	VAR robtarget Openhole_1322 := [[444.74, -6.64, 181.61], [-0.056167, 0.704873, 0.706652, -0.025359], [0,0,0,0], [9E9, 9E9, 9E9, 9E9, 9E9, 9E9]];
	VAR robtarget Openhole_1323 := [[441.88, -4.7, 182.09], [-0.072208, 0.70341, 0.706763, -0.02205], [0,0,0,0], [9E9, 9E9, 9E9, 9E9, 9E9, 9E9]];
	VAR robtarget Openhole_1324 := [[439.03, -2.77, 182.68], [-0.088015, 0.701608, 0.706859, -0.018705], [0,0,0,0], [9E9, 9E9, 9E9, 9E9, 9E9, 9E9]];
	VAR robtarget Openhole_1325 := [[445.19, -0.91, 181.79], [-0.073661, 0.70326, 0.70561, -0.045986], [0,0,0,0], [9E9, 9E9, 9E9, 9E9, 9E9, 9E9]];
	VAR robtarget Openhole_1326 := [[446.14, -0.63, 181.63], [-0.07136, 0.703497, 0.705328, -0.050126], [0,0,0,0], [9E9, 9E9, 9E9, 9E9, 9E9, 9E9]];
	VAR robtarget Openhole_1327 := [[447.09, -0.38, 181.47], [-0.06898, 0.703734, 0.705025, -0.054215], [0,0,0,0], [9E9, 9E9, 9E9, 9E9, 9E9, 9E9]];
	VAR robtarget Openhole_1328 := [[447.57, -0.24, 181.38], [-0.067831, 0.703846, 0.704863, -0.05628], [0,0,0,0], [9E9, 9E9, 9E9, 9E9, 9E9, 9E9]];
	VAR robtarget Openhole_1329 := [[448.04, -0.13, 181.3], [-0.066601, 0.703963, 0.7047, -0.058297], [0,0,0,0], [9E9, 9E9, 9E9, 9E9, 9E9, 9E9]];
	VAR robtarget Openhole_1330 := [[448.52, 0, 181.21], [-0.065406, 0.704075, 0.704528, -0.060332], [0,0,0,0], [9E9, 9E9, 9E9, 9E9, 9E9, 9E9]];
	VAR robtarget Openhole_1331 := [[449.49, 0.16, 181.03], [-0.062643, 0.704327, 0.70419, -0.064159], [0,0,0,0], [9E9, 9E9, 9E9, 9E9, 9E9, 9E9]];
	VAR robtarget Openhole_1332 := [[450.47, 0.12, 180.85], [-0.059198, 0.704624, 0.703889, -0.067379], [0,0,0,0], [9E9, 9E9, 9E9, 9E9, 9E9, 9E9]];
	VAR robtarget Openhole_1333 := [[451.43, -0.1, 180.68], [-0.055192, 0.70495, 0.703646, -0.069869], [0,0,0,0], [9E9, 9E9, 9E9, 9E9, 9E9, 9E9]];
	VAR robtarget Openhole_1334 := [[451.9, -0.27, 180.6], [-0.053064, 0.705113, 0.703545, -0.070885], [0,0,0,0], [9E9, 9E9, 9E9, 9E9, 9E9, 9E9]];
	VAR robtarget Openhole_1335 := [[452.84, -0.58, 180.44], [-0.048861, 0.705417, 0.703324, -0.07304], [0,0,0,0], [9E9, 9E9, 9E9, 9E9, 9E9, 9E9]];
	VAR robtarget Openhole_1336 := [[453.8, -0.8, 180.28], [-0.044856, 0.705683, 0.703059, -0.075549], [0,0,0,0], [9E9, 9E9, 9E9, 9E9, 9E9, 9E9]];
	VAR robtarget Openhole_1337 := [[454.76, -0.99, 180.12], [-0.040922, 0.705922, 0.702773, -0.078167], [0,0,0,0], [9E9, 9E9, 9E9, 9E9, 9E9, 9E9]];
	VAR robtarget Openhole_1338 := [[457.2, -1.38, 179.73], [-0.031334, 0.706412, 0.701973, -0.085051], [0,0,0,0], [9E9, 9E9, 9E9, 9E9, 9E9, 9E9]];
	VAR robtarget Openhole_1339 := [[459.17, -1.56, 179.41], [-0.02402, 0.706699, 0.70123, -0.090973], [0,0,0,0], [9E9, 9E9, 9E9, 9E9, 9E9, 9E9]];
	VAR robtarget Openhole_1340 := [[460.16, -1.6, 179.25], [-0.020505, 0.706809, 0.700821, -0.094075], [0,0,0,0], [9E9, 9E9, 9E9, 9E9, 9E9, 9E9]];
	VAR robtarget Openhole_1341 := [[461.14, -1.61, 179.08], [-0.017095, 0.7069, 0.700384, -0.097271], [0,0,0,0], [9E9, 9E9, 9E9, 9E9, 9E9, 9E9]];
	VAR robtarget Openhole_1342 := [[461.64, -1.61, 179], [-0.01542, 0.706939, 0.700158, -0.098891], [0,0,0,0], [9E9, 9E9, 9E9, 9E9, 9E9, 9E9]];
	VAR robtarget Openhole_1343 := [[467.04, -1.32, 178.04], [0.002033, 0.707104, 0.697314, -0.117272], [0,0,0,0], [9E9, 9E9, 9E9, 9E9, 9E9, 9E9]];
	VAR robtarget Openhole_1344 := [[474.41, -0.89, 176.69], [0.025407, 0.70665, 0.692796, -0.141541], [0,0,0,0], [9E9, 9E9, 9E9, 9E9, 9E9, 9E9]];
	VAR robtarget Openhole_1345 := [[476.87, -0.86, 176.25], [0.033467, 0.706314, 0.691219, -0.149049], [0,0,0,0], [9E9, 9E9, 9E9, 9E9, 9E9, 9E9]];
	VAR robtarget Openhole_1346 := [[477.36, -0.86, 176.16], [0.035102, 0.706235, 0.690903, -0.150508], [0,0,0,0], [9E9, 9E9, 9E9, 9E9, 9E9, 9E9]];
	VAR robtarget Openhole_1347 := [[482.78, -1.08, 175.28], [0.053469, 0.705082, 0.687432, -0.165642], [0,0,0,0], [9E9, 9E9, 9E9, 9E9, 9E9, 9E9]];
	VAR robtarget Openhole_1348 := [[488.7, -1.64, 174.47], [0.073993, 0.703225, 0.683703, -0.180416], [0,0,0,0], [9E9, 9E9, 9E9, 9E9, 9E9, 9E9]];
	VAR robtarget Openhole_1349 := [[495.1, -2.58, 173.82], [0.096389, 0.700506, 0.679807, -0.194582], [0,0,0,0], [9E9, 9E9, 9E9, 9E9, 9E9, 9E9]];
	VAR robtarget Openhole_1350 := [[495.59, -2.66, 173.77], [0.098105, 0.700268, 0.679515, -0.1956], [0,0,0,0], [9E9, 9E9, 9E9, 9E9, 9E9, 9E9]];
	VAR robtarget Openhole_1351 := [[495.54, -3.95, 174.35], [0.101813, 0.699739, 0.680628, -0.191692], [0,0,0,0], [9E9, 9E9, 9E9, 9E9, 9E9, 9E9]];
	VAR robtarget Openhole_1352 := [[488.63, -3.04, 175.01], [0.078064, 0.702785, 0.684848, -0.176019], [0,0,0,0], [9E9, 9E9, 9E9, 9E9, 9E9, 9E9]];
	VAR robtarget Openhole_1353 := [[482.7, -2.51, 175.76], [0.057702, 0.704748, 0.688538, -0.160983], [0,0,0,0], [9E9, 9E9, 9E9, 9E9, 9E9, 9E9]];
	VAR robtarget Openhole_1354 := [[477.26, -2.32, 176.57], [0.039419, 0.706007, 0.691941, -0.145665], [0,0,0,0], [9E9, 9E9, 9E9, 9E9, 9E9, 9E9]];
	VAR robtarget Openhole_1355 := [[476.77, -2.31, 176.65], [0.037788, 0.706096, 0.692249, -0.144192], [0,0,0,0], [9E9, 9E9, 9E9, 9E9, 9E9, 9E9]];
	VAR robtarget Openhole_1356 := [[476.28, -2.32, 176.73], [0.036172, 0.706181, 0.692558, -0.142699], [0,0,0,0], [9E9, 9E9, 9E9, 9E9, 9E9, 9E9]];
	VAR robtarget Openhole_1357 := [[470.37, -2.56, 177.73], [0.017259, 0.706896, 0.696188, -0.123785], [0,0,0,0], [9E9, 9E9, 9E9, 9E9, 9E9, 9E9]];
	VAR robtarget Openhole_1358 := [[462.5, -3.12, 179.05], [-0.007511, 0.707067, 0.700456, -0.096756], [0,0,0,0], [9E9, 9E9, 9E9, 9E9, 9E9, 9E9]];
	VAR robtarget Openhole_1359 := [[461.51, -3.15, 179.2], [-0.010776, 0.707025, 0.700907, -0.093428], [0,0,0,0], [9E9, 9E9, 9E9, 9E9, 9E9, 9E9]];
	VAR robtarget Openhole_1360 := [[461.01, -3.16, 179.28], [-0.012455, 0.706997, 0.701123, -0.0918], [0,0,0,0], [9E9, 9E9, 9E9, 9E9, 9E9, 9E9]];
	VAR robtarget Openhole_1361 := [[460.52, -3.16, 179.35], [-0.014142, 0.706965, 0.701333, -0.090176], [0,0,0,0], [9E9, 9E9, 9E9, 9E9, 9E9, 9E9]];
	VAR robtarget Openhole_1362 := [[459.53, -3.13, 179.5], [-0.017599, 0.706888, 0.701734, -0.087], [0,0,0,0], [9E9, 9E9, 9E9, 9E9, 9E9, 9E9]];
	VAR robtarget Openhole_1363 := [[458.54, -3.07, 179.65], [-0.021156, 0.70679, 0.70211, -0.083916], [0,0,0,0], [9E9, 9E9, 9E9, 9E9, 9E9, 9E9]];
	VAR robtarget Openhole_1364 := [[454.62, -2.55, 180.22], [-0.036285, 0.706175, 0.703373, -0.07257], [0,0,0,0], [9E9, 9E9, 9E9, 9E9, 9E9, 9E9]];
	VAR robtarget Openhole_1365 := [[451.22, -1.9, 180.75], [-0.049988, 0.705338, 0.704274, -0.063233], [0,0,0,0], [9E9, 9E9, 9E9, 9E9, 9E9, 9E9]];
	VAR robtarget Openhole_1366 := [[450.73, -1.83, 180.83], [-0.051876, 0.705201, 0.704401, -0.061803], [0,0,0,0], [9E9, 9E9, 9E9, 9E9, 9E9, 9E9]];
	VAR robtarget Openhole_1367 := [[450.24, -1.78, 180.91], [-0.053711, 0.705064, 0.70453, -0.06031], [0,0,0,0], [9E9, 9E9, 9E9, 9E9, 9E9, 9E9]];
	VAR robtarget Openhole_1368 := [[449.75, -1.74, 180.99], [-0.055508, 0.704925, 0.70466, -0.058768], [0,0,0,0], [9E9, 9E9, 9E9, 9E9, 9E9, 9E9]];
	VAR robtarget Openhole_1369 := [[449.26, -1.74, 181.08], [-0.057188, 0.70479, 0.704797, -0.057102], [0,0,0,0], [9E9, 9E9, 9E9, 9E9, 9E9, 9E9]];
	VAR robtarget Openhole_1370 := [[448.77, -1.75, 181.16], [-0.05882, 0.704656, 0.704934, -0.055386], [0,0,0,0], [9E9, 9E9, 9E9, 9E9, 9E9, 9E9]];
	VAR robtarget Openhole_1371 := [[448.27, -1.79, 181.24], [-0.060366, 0.704525, 0.705073, -0.05359], [0,0,0,0], [9E9, 9E9, 9E9, 9E9, 9E9, 9E9]];
	VAR robtarget Openhole_1372 := [[447.78, -1.85, 181.32], [-0.061814, 0.7044, 0.705213, -0.051717], [0,0,0,0], [9E9, 9E9, 9E9, 9E9, 9E9, 9E9]];
	VAR robtarget Openhole_1373 := [[447.3, -1.93, 181.4], [-0.063211, 0.704276, 0.705351, -0.049802], [0,0,0,0], [9E9, 9E9, 9E9, 9E9, 9E9, 9E9]];
	VAR robtarget Openhole_1374 := [[446.81, -2.01, 181.48], [-0.064564, 0.704153, 0.705486, -0.047856], [0,0,0,0], [9E9, 9E9, 9E9, 9E9, 9E9, 9E9]];
	VAR robtarget Openhole_1375 := [[445.84, -2.22, 181.63], [-0.067123, 0.703914, 0.705745, -0.04386], [0,0,0,0], [9E9, 9E9, 9E9, 9E9, 9E9, 9E9]];
	VAR robtarget Openhole_1376 := [[444.89, -2.47, 181.77], [-0.069529, 0.70368, 0.705988, -0.039766], [0,0,0,0], [9E9, 9E9, 9E9, 9E9, 9E9, 9E9]];
	VAR robtarget Openhole_1377 := [[438.19, -4.32, 182.64], [-0.085686, 0.701896, 0.707026, -0.01071], [0,0,0,0], [9E9, 9E9, 9E9, 9E9, 9E9, 9E9]];
	VAR robtarget Openhole_1378 := [[437.22, -4.54, 182.75], [-0.088153, 0.70159, 0.707075, -0.006674], [0,0,0,0], [9E9, 9E9, 9E9, 9E9, 9E9, 9E9]];
	VAR robtarget Openhole_1379 := [[431.67, -6.99, 183.11], [-0.098095, 0.700269, 0.706815, 0.020318], [0,0,0,0], [9E9, 9E9, 9E9, 9E9, 9E9, 9E9]];
	VAR robtarget Openhole_1380 := [[438.07, -6.03, 182.47], [-0.080435, 0.702517, 0.707092, -0.004596], [0,0,0,0], [9E9, 9E9, 9E9, 9E9, 9E9, 9E9]];
	VAR robtarget Openhole_1381 := [[444.39, -4.68, 181.75], [-0.063882, 0.704215, 0.70644, -0.030694], [0,0,0,0], [9E9, 9E9, 9E9, 9E9, 9E9, 9E9]];
	VAR robtarget Openhole_1382 := [[444.87, -4.57, 181.68], [-0.06262, 0.704329, 0.70635, -0.032715], [0,0,0,0], [9E9, 9E9, 9E9, 9E9, 9E9, 9E9]];
	VAR robtarget Openhole_1383 := [[445.84, -4.38, 181.56], [-0.060005, 0.704556, 0.706154, -0.036695], [0,0,0,0], [9E9, 9E9, 9E9, 9E9, 9E9, 9E9]];
	VAR robtarget Openhole_1384 := [[446.33, -4.29, 181.49], [-0.058643, 0.704671, 0.70605, -0.038646], [0,0,0,0], [9E9, 9E9, 9E9, 9E9, 9E9, 9E9]];
